Fanuc TP program (LS listing): OP5_LRG_SEQCHNG_AIR_BASE.LS

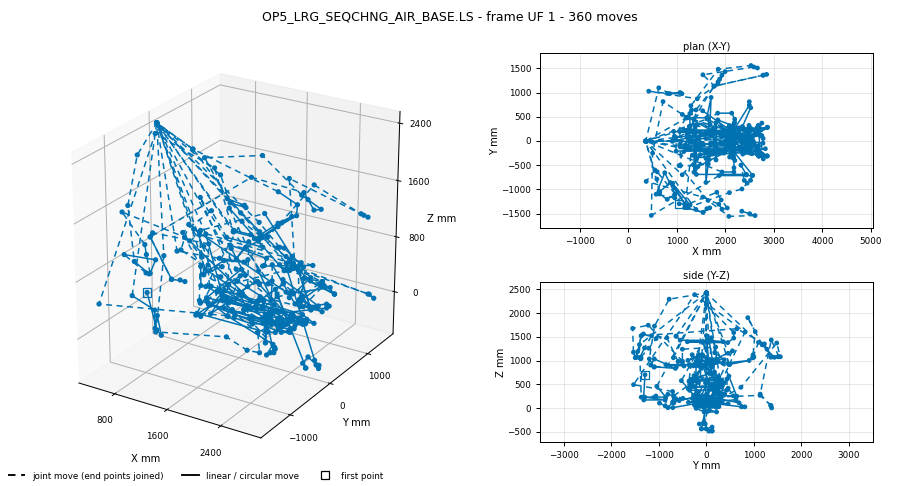
[picture p0: tool path of OP5_LRG_SEQCHNG_AIR_BASE.LS in frame UF 1, 360 of 361 moves have a stored position in this frame; points joined in program order, loops and branches not executed]
/PROG  OP5_LRG_SEQCHNG_AIR_BASE
/ATTR
OWNER		= MNEDITOR;
COMMENT		= "Large Main Air";
PROG_SIZE	= 92875;
CREATE		= DATE 26-02-26  TIME 08:30:24;
MODIFIED	= DATE 26-02-26  TIME 08:30:24;
FILE_NAME	= OP5_LRG_;
VERSION		= 0;
LINE_COUNT	= 2422;
MEMORY_SIZE	= 93511;
PROTECT		= READ_WRITE;
TCD:  STACK_SIZE	= 0,
      TASK_PRIORITY	= 50,
      TIME_SLICE	= 0,
      BUSY_LAMP_OFF	= 0,
      ABORT_REQUEST	= 0,
      PAUSE_REQUEST	= 0;
DEFAULT_GROUP	= 1,1,*,*,*;
CONTROL_CODE	= 00000000 00000000;
/APPL
  ARC Welding Equipment : 1,*,*,*,*;

MPAS ;
MPAS_NUM_PASSES        : 0;
MPAS_LAST_PASS         : 0;
MPAS_CURRENT_PASS      : 0;
MPAS_STATUS_PASS       : 0;
/MN
   1:  !********** WAR HAMMER ********** ;
   2:  !*------- FRAME LARGE ----------* ;
   3:  !*-- WELD SEQUENCE CHANGE 2026--* ;
   4:  !*------- FR500 CELL: A --------* ;
   5:  !******************************** ;
   6:   ;
   7:  CALL HOME    ;
   8:  UFRAME_NUM=1 ;
   9:  DO[17:OFF:WIRE BRAKE]=OFF ;
  10:   ;
  11:  !********POSITIONER MOVE******** ;
  12:J P[1] 85% CNT40    ;
  13:   ;
  14:L P[3] 1000mm/sec CNT40    ;
  15:   ;
  16:  !FR50L1000 ;
  17:  IF R[15]=1002,CALL TECH_HOLD ;
  18:   ;
  19:  !TO SKIP FRONT BUMPER WELDS ;
  20:  CALL ARC_DISABLE_FRONT_BMPR_LRG(0) ;
  21:   ;
  22:   ;
 2:  --eg:PASTE (FR50L1000) ;
  29:   ;
  30:   ;
  31:   ;
  32:L P[8] 800mm/sec CNT30    ;
  33:   ;
  34:L P[9] 1000mm/sec CNT30    ;
  35:   ;
  36:   ;
  37:  !FR50L1001 ;
  38:  IF R[15]=1003,CALL TECH_HOLD ;
  39:   ;
  40:   ;
  41:   ;
 2:  --eg:PASTE (FR50L1001) ;
  48:   ;
  49:   ;
  50:L P[12] 1000mm/sec CNT100    ;
  51:   ;
  52:   ;
  53:  !FR50L1002 ;
  54:  IF R[15]=1004,CALL TECH_HOLD ;
  55:   ;
  56:   ;
  57:L P[13] 1000mm/sec CNT70    ;
  58:   ;
  59:   ;
 2:  --eg:PASTE (FR50L1002) ;
  66:   ;
  67:   ;
  68:  CALL ARC_DISABLE_FRONT_BMPR_LRG(1) ;
  69:   ;
  70:L P[16] 1000mm/sec CNT100    ;
  71:   ;
  72:  !HOME ;
  73:J P[4] 70% CNT30    ;
  74:   ;
  75:  !********POSITIONER MOVE******** ;
  76:J P[17] 85% CNT30    ;
  77:   ;
  78:J P[18] 50% CNT100    ;
  79:   ;
  80:L P[19] 1000mm/sec CNT100    ;
  81:   ;
  82:   ;
  83:  !FR50L1003 ;
  84:  IF R[15]=1005,CALL TECH_HOLD ;
  85:   ;
  86:   ;
  87:L P[20] 1000mm/sec CNT25    ;
  88:   ;
  89:   ;
 2:  --eg:PASTE (FR50L1003) ;
  97:   ;
  98:   ;
  99:L P[24] 1000mm/sec CNT30    ;
 100:   ;
 101:   ;
 102:  !FR50L1010 ;
 103:  IF R[15]=1012,CALL TECH_HOLD ;
 104:   ;
 105:   ;
 106:L P[25] 1000mm/sec CNT30    ;
 107:   ;
 108:   ;
 2:  --eg:PASTE (FR50L1010) ;
 116:   ;
 117:   ;
 118:L P[29] 1000mm/sec CNT25    ;
 119:   ;
 120:   ;
 121:  !FR50L1020 ;
 122:  IF R[15]=1022,CALL TECH_HOLD ;
 123:   ;
 124:   ;
 125:J P[30] 50% CNT25    ;
 126:   ;
 127:   ;
 2:  --eg:PASTE (FR50L1020) ;
 134:   ;
 135:   ;
 136:L P[33] 1000mm/sec CNT30    ;
 137:   ;
 138:L P[34] 1000mm/sec CNT30    ;
 139:   ;
 140:   ;
 141:  !FR50L1030 ;
 142:  IF R[15]=1032,CALL TECH_HOLD ;
 143:   ;
 144:   ;
 145:   ;
 2:  --eg:PASTE (FR50L1030) ;
 152:   ;
 153:   ;
 154:L P[37] 1000mm/sec CNT50    ;
 155:   ;
 156:J P[38] 50% CNT50    ;
 157:   ;
 158:L P[39] 1000mm/sec CNT25    ;
 159:   ;
 160:   ;
 161:  !FR50L1040 ;
 162:  IF R[15]=1042,CALL TECH_HOLD ;
 163:   ;
 164:   ;
 165:   ;
 2:  --eg:PASTE (FR50L1040) ;
 170:   ;
 171:   ;
 172:L P[42] 1000mm/sec CNT30    ;
 173:   ;
 174:L P[43] 1000mm/sec CNT70    ;
 175:   ;
 176:J P[44] 50% CNT50    ;
 177:   ;
 178:L P[45] 1000mm/sec CNT30    ;
 179:   ;
 180:   ;
 181:  !FR50L1050 ;
 182:  IF R[15]=1052,CALL TECH_HOLD ;
 183:   ;
 184:   ;
 185:   ;
 2:  --eg:PASTE (FR50L1050) ;
 190:   ;
 191:   ;
 192:L P[48] 1000mm/sec CNT80    ;
 193:   ;
 194:J P[49] 50% CNT25    ;
 195:   ;
 196:L P[50] 1000mm/sec CNT25    ;
 197:   ;
 198:   ;
 199:  !FR50L1060 ;
 200:  IF R[15]=1062,CALL TECH_HOLD ;
 201:   ;
 202:   ;
 203:   ;
 2:  --eg:PASTE (FR50L1060) ;
 208:   ;
 209:   ;
 210:L P[53] 500mm/sec CNT100    ;
 211:   ;
 212:L P[54] 1500mm/sec CNT35    ;
 213:   ;
 214:J P[55] 50% CNT30    ;
 215:   ;
 216:L P[56] 1000mm/sec CNT30    ;
 217:   ;
 218:   ;
 219:  !FR50L1070 ;
 220:  IF R[15]=1072,CALL TECH_HOLD ;
 221:   ;
 222:   ;
 223:   ;
 2:  --eg:PASTE (FR50L1070) ;
 230:   ;
 231:   ;
 232:L P[59] 1000mm/sec CNT100    ;
 233:   ;
 234:L P[60] 1000mm/sec CNT80    ;
 235:   ;
 236:   ;
 237:  !FR50L1080 ;
 238:  IF R[15]=1082,CALL TECH_HOLD ;
 239:   ;
 240:   ;
 241:   ;
 2:  --eg:PASTE (FR50L1080) ;
 248:   ;
 249:   ;
 250:J P[63] 30% CNT100    ;
 251:   ;
 252:J P[64] 50% CNT100    ;
 253:   ;
 254:L P[65] 1000mm/sec CNT80    ;
 255:   ;
 256:   ;
 257:  !FR50L1090 ;
 258:  IF R[15]=1092,CALL TECH_HOLD ;
 259:  !10MM PASS ;
 260:   ;
 261:   ;
 262:   ;
 2:  --eg:PASTE (FR50L1090) ;
 272:   ;
 273:   ;
 274:J P[72] 16% CNT25    ;
 275:   ;
 276:J P[74] 50% CNT25    ;
 277:   ;
 278:L P[75] 1000mm/sec CNT25    ;
 279:   ;
 280:   ;
 281:  !FR50L1100 ;
 282:  IF R[15]=1102,CALL TECH_HOLD ;
 283:   ;
 284:   ;
 285:   ;
 2:  --eg:PASTE (FR50L1100) ;
 295:   ;
 296:   ;
 297:J P[82] 50% CNT10    ;
 298:   ;
 299:J P[83] 50% CNT80    ;
 300:   ;
 301:L P[84] 1000mm/sec CNT25    ;
 302:   ;
 303:   ;
 304:  !FR50L1110MP1 ;
 305:  IF R[15]=1112,CALL TECH_HOLD ;
 306:   ;
 307:   ;
 308:  MP Offset  PR[3] RPM[1] ;
 309:   ;
 2:  --eg:PASTE (FR50L1110MP1) ;
 317:   ;
 318:  MP Offset End ;
 319:   ;
 320:J P[91] 40% CNT10    ;
 321:   ;
 322:J P[92] 50% CNT30    ;
 323:   ;
 324:L P[93] 1000mm/sec CNT25    ;
 325:   ;
 326:   ;
 327:  !FR50M1110MP2 ;
 328:   ;
 329:   ;
 330:  MP Offset  PR[4] RPM[1] ;
 331:   ;
 2:  --eg:PASTE (FR50M1110MP2) ;
 339:   ;
 340:  MP Offset End ;
 341:   ;
 342:J P[100] 50% CNT25    ;
 343:   ;
 344:J P[102] 50% CNT25    ;
 345:   ;
 346:L P[103] 1000mm/sec CNT25    ;
 347:   ;
 348:   ;
 349:  !FR50L1120MP3 ;
 350:  IF R[15]=1122,CALL TECH_HOLD ;
 351:   ;
 352:   ;
 353:  MP Offset  PR[1] RPM[2] ;
 354:   ;
 2:  --eg:PASTE (FR50L1120MP3) ;
 362:   ;
 363:  MP Offset End ;
 364:   ;
 365:J P[110] 50% CNT25    ;
 366:   ;
 367:J P[111] 50% CNT25    ;
 368:   ;
 369:L P[112] 1000mm/sec CNT25    ;
 370:   ;
 371:   ;
 372:  !FR501130MP4 ;
 373:   ;
 374:   ;
 375:  MP Offset  PR[2] RPM[2] ;
 376:   ;
 2:  --eg:PASTE (FR501130MP4) ;
 384:   ;
 385:  MP Offset End ;
 386:   ;
 387:J P[119] 50% CNT25    ;
 388:   ;
 389:J P[121] 50% CNT25    ;
 390:   ;
 391:L P[122] 1000mm/sec CNT25    ;
 392:   ;
 393:   ;
 394:  !FR50L1140 ;
 395:  IF R[15]=1142,CALL TECH_HOLD ;
 396:   ;
 397:   ;
 398:   ;
 2:  --eg:PASTE (FR50L1140) ;
 404:   ;
 405:   ;
 406:L P[127] 1000mm/sec CNT25    ;
 407:   ;
 408:J P[128] 50% CNT25    ;
 409:   ;
 410:   ;
 411:  !FR50L1141 ;
 412:  IF R[15]=1143,CALL TECH_HOLD ;
 413:   ;
 414:   ;
 415:   ;
 2:  --eg:PASTE (FR50L1141) ;
 421:   ;
 422:   ;
 423:L P[133] 1000mm/sec CNT25    ;
 424:   ;
 425:L P[134] 1000mm/sec CNT25    ;
 426:   ;
 427:J P[135] 50% CNT25    ;
 428:   ;
 429:L P[136] 1000mm/sec CNT50    ;
 430:   ;
 431:   ;
 432:  !FR50L1150 ;
 433:  IF R[15]=1152,CALL TECH_HOLD ;
 434:   ;
 435:   ;
 436:   ;
 2:  --eg:PASTE (FR50L1150) ;
 443:   ;
 444:   ;
 445:L P[139] 1000mm/sec CNT100    ;
 446:   ;
 447:L P[140] 1000mm/sec CNT50    ;
 448:   ;
 449:   ;
 450:  !FR50L1160 ;
 451:  IF R[15]=1162,CALL TECH_HOLD ;
 452:   ;
 453:   ;
 2:  --eg:PASTE (FR50L1160) ;
 460:   ;
 461:   ;
 462:L P[143] 1000mm/sec CNT30    ;
 463:   ;
 464:  !********POSITIONER MOVE******** ;
 465:J P[144] 85% CNT30    ;
 466:   ;
 467:L P[145] 1000mm/sec CNT100    ;
 468:   ;
 469:   ;
 470:  !FR50L1170 ;
 471:  IF R[15]=1172,CALL TECH_HOLD ;
 472:   ;
 473:   ;
 474:   ;
 2:  --eg:PASTE (FR50L1170) ;
 481:   ;
 482:   ;
 483:L P[148] 1000mm/sec CNT100    ;
 484:   ;
 485:L P[149] 1500mm/sec CNT100    ;
 486:   ;
 487:   ;
 488:  !FR50L1180 ;
 489:  IF R[15]=1182,CALL TECH_HOLD ;
 490:   ;
 491:   ;
 492:   ;
 2:  --eg:PASTE (FR50L1180) ;
 499:   ;
 500:   ;
 501:L P[152] 1000mm/sec CNT100    ;
 502:   ;
 503:  !HOME ;
 504:J P[7] 100% CNT30    ;
 505:   ;
 506:  !********POSITIONER MOVE******** ;
 507:J P[153] 80% CNT30    ;
 508:   ;
 509:J P[154] 50% CNT100    ;
 510:   ;
 511:L P[155] 1000mm/sec CNT25    ;
 512:   ;
 513:   ;
 514:  !FR50L1210 ;
 515:  IF R[15]=1212,CALL TECH_HOLD ;
 516:   ;
 517:   ;
 518:   ;
 2:  --eg:PASTE (FR50L1210) ;
 526:   ;
 527:   ;
 528:L P[159] 1000mm/sec CNT25    ;
 529:   ;
 530:L P[160] 1000mm/sec CNT25    ;
 531:   ;
 532:   ;
 533:  !FR50L1220 ;
 534:  IF R[15]=1222,CALL TECH_HOLD ;
 535:   ;
 536:   ;
 537:   ;
 2:  --eg:PASTE (FR50L1220) ;
 544:   ;
 545:   ;
 546:L P[163] 1000mm/sec CNT80    ;
 547:   ;
 548:L P[164] 1200mm/sec CNT25    ;
 549:   ;
 550:   ;
 551:  !FR50L1230 ;
 552:  IF R[15]=1232,CALL TECH_HOLD ;
 553:   ;
 554:   ;
 555:   ;
 2:  --eg:PASTE (FR50L1230) ;
 562:   ;
 563:   ;
 564:L P[167] 1000mm/sec CNT25    ;
 565:   ;
 566:L P[168] 1000mm/sec CNT25    ;
 567:   ;
 568:   ;
 569:  !FR50L1240 ;
 570:  IF R[15]=1242,CALL TECH_HOLD ;
 571:   ;
 572:   ;
 573:   ;
 2:  --eg:PASTE (FR50L1240) ;
 581:   ;
 582:   ;
 583:L P[172] 1000mm/sec CNT25    ;
 584:   ;
 585:L P[173] 1000mm/sec CNT100    ;
 586:   ;
 587:  !HOME ;
 588:J P[116] 100% CNT100    ;
 589:   ;
 590:   ;
 591:  !********POSITIONER MOVE******** ;
 592:J P[174] 85% FINE    ;
 593:   ;
 594:  CALL T_CLEAN    ;
 595:   ;
 596:J P[175] 50% CNT35    ;
 597:   ;
 598:L P[176] 1000mm/sec CNT25    ;
 599:   ;
 600:   ;
 601:  !FR50L1250 ;
 602:  IF R[15]=1252,CALL TECH_HOLD ;
 603:   ;
 604:   ;
 605:   ;
 2:  --eg:PASTE (FR50L1250) ;
 614:   ;
 615:   ;
 616:L P[181] 1000mm/sec CNT100    ;
 617:   ;
 618:J P[182] 50% CNT100    ;
 619:   ;
 620:L P[184] 500mm/sec CNT100    ;
 621:   ;
 622:   ;
 623:  !FR50L1260 ;
 624:  IF R[15]=1262,CALL TECH_HOLD ;
 625:   ;
 626:   ;
 627:   ;
 2:  --eg:PASTE (FR50L1260) ;
 636:   ;
 637:   ;
 638:L P[189] 1000mm/sec CNT25    ;
 639:   ;
 640:J P[190] 50% CNT25    ;
 641:   ;
 642:L P[191] 1000mm/sec CNT25    ;
 643:   ;
 644:   ;
 645:  !FR50L1270 ;
 646:  IF R[15]=1272,CALL TECH_HOLD ;
 647:   ;
 648:   ;
 649:   ;
 2:  --eg:PASTE (FR50L1270) ;
 657:   ;
 658:   ;
 659:L P[195] 1000mm/sec CNT80    ;
 660:   ;
 661:L P[196] 1000mm/sec CNT100    ;
 662:   ;
 663:   ;
 664:  !FR50L1280 ;
 665:  IF R[15]=1282,CALL TECH_HOLD ;
 666:   ;
 667:   ;
 668:   ;
 2:  --eg:PASTE (FR50L1280) ;
 676:   ;
 677:   ;
 678:L P[200] 1000mm/sec CNT25    ;
 679:   ;
 680:J P[201] 50% CNT25    ;
 681:   ;
 682:L P[202] 1000mm/sec CNT25    ;
 683:   ;
 684:   ;
 685:  !FR50L1290 ;
 686:  IF R[15]=1292,CALL TECH_HOLD ;
 687:   ;
 688:   ;
 689:   ;
 2:  --eg:PASTE (FR50L1290) ;
 697:   ;
 698:   ;
 699:L P[206] 1000mm/sec CNT100    ;
 700:   ;
 701:L P[207] 1000mm/sec CNT100    ;
 702:   ;
 703:   ;
 704:  !FR50L1300 ;
 705:  IF R[15]=1302,CALL TECH_HOLD ;
 706:   ;
 707:   ;
 708:   ;
 2:  --eg:PASTE (FR50L1300) ;
 715:   ;
 716:   ;
 717:L P[210] 1000mm/sec CNT100    ;
 718:   ;
 719:L P[211] 1000mm/sec CNT100    ;
 720:   ;
 721:   ;
 722:  !FR50L1310 ;
 723:  IF R[15]=1312,CALL TECH_HOLD ;
 724:   ;
 725:   ;
 726:   ;
 2:  --eg:PASTE (FR50L1310) ;
 733:   ;
 734:   ;
 735:L P[214] 1000mm/sec CNT100    ;
 736:   ;
 737:L P[215] 1000mm/sec CNT100    ;
 738:   ;
 739:   ;
 740:  !FR50L1320 ;
 741:  IF R[15]=1322,CALL TECH_HOLD ;
 742:   ;
 743:   ;
 744:   ;
 2:  --eg:PASTE (FR50L1320) ;
 752:   ;
 753:   ;
 754:L P[219] 1000mm/sec CNT100    ;
 755:   ;
 756:L P[220] 1000mm/sec CNT100    ;
 757:   ;
 758:J P[73] 50% CNT30    ;
 759:   ;
 760:  !********POSITIONER MOVE******** ;
 761:J P[86] 100% CNT30    ;
 762:   ;
 763:  !FR50L1330 ;
 764:  IF R[15]=1332,CALL TECH_HOLD ;
 765:   ;
 766:   ;
 767:J P[327] 40% CNT10    ;
 768:   ;
 769:   ;
 2:  --eg:PASTE (FR50L1330) ;
 774:   ;
 775:   ;
 776:J P[85] 50% CNT30    ;
 777:   ;
 778:L P[233] 1000mm/sec CNT25    ;
 779:   ;
 780:  !********POSITIONER MOVE******** ;
 781:J P[225] 80% CNT20    ;
 782:   ;
 783:   ;
 784:   ;
 785:  !FR50L1340 ;
 786:  IF R[15]=1342,CALL TECH_HOLD ;
 787:   ;
 788:   ;
 789:   ;
 2:  --eg:PASTE (FR50L1340) ;
 794:   ;
 795:   ;
 796:   ;
 797:  !FR50L1350 ;
 798:  IF R[15]=1352,CALL TECH_HOLD ;
 799:   ;
 800:   ;
 801:   ;
 2:  --eg:PASTE (FR50L1350) ;
 806:   ;
 807:   ;
 808:L P[230] 1000mm/sec CNT25    ;
 809:   ;
 810:  !HOME ;
 811:J P[117] 100% CNT50    ;
 812:   ;
 813:  !********POSITIONER MOVE******** ;
 814:J P[768] 85% CNT25    ;
 815:   ;
 816:L P[234] 1000mm/sec CNT25    ;
 817:   ;
 818:J P[235] 50% CNT25    ;
 819:   ;
 820:   ;
 821:  !FR50L1380 ;
 822:  IF R[15]=1382,CALL TECH_HOLD ;
 823:   ;
 824:   ;
 825:   ;
 2:  --eg:PASTE (FR50L1380) ;
 834:   ;
 835:   ;
 836:L P[240] 800mm/sec CNT2    ;
 837:   ;
 838:L P[241] 800mm/sec CNT25    ;
 839:   ;
 840:  !********POSITIONER MOVE******** ;
 841:J P[242] 75% CNT5    ;
 842:   ;
 843:L P[243] 1000mm/sec CNT25    ;
 844:   ;
 845:   ;
 846:  !FR50L1390 ;
 847:  IF R[15]=1392,CALL TECH_HOLD ;
 848:   ;
 849:   ;
 2:  --eg:PASTE (FR50L1390) ;
 856:   ;
 857:   ;
 858:L P[248] 1000mm/sec CNT25    ;
 859:   ;
 860:L P[249] 1000mm/sec CNT25    ;
 861:   ;
 862:   ;
 863:  !FR50L1400 ;
 864:  IF R[15]=1402,CALL TECH_HOLD ;
 865:   ;
 866:   ;
 867:   ;
 2:  --eg:PASTE (FR50L1400) ;
 874:   ;
 875:   ;
 876:L P[252] 1000mm/sec CNT25    ;
 877:   ;
 878:   ;
 879:  !FR50L1410 ;
 880:  IF R[15]=1412,CALL TECH_HOLD ;
 881:   ;
 882:   ;
 883:   ;
 2:  --eg:PASTE (FR50L1410) ;
 891:   ;
 892:   ;
 893:L P[256] 1000mm/sec CNT25    ;
 894:   ;
 895:   ;
 896:  !FR50L1420 ;
 897:  IF R[15]=1422,CALL TECH_HOLD ;
 898:   ;
 899:   ;
 900:   ;
 2:  --eg:PASTE (FR50L1420) ;
 908:   ;
 909:   ;
 910:L P[260] 1000mm/sec CNT25    ;
 911:   ;
 912:L P[261] 1000mm/sec CNT25    ;
 913:   ;
 914:   ;
 915:  !FR50L1430 ;
 916:  IF R[15]=1432,CALL TECH_HOLD ;
 917:   ;
 918:   ;
 919:   ;
 2:  --eg:PASTE (FR50L1430) ;
 925:   ;
 926:   ;
 927:L P[265] 1000mm/sec CNT25    ;
 928:   ;
 929:   ;
 930:  !FR50L1431 ;
 931:  IF R[15]=1433,CALL TECH_HOLD ;
 932:   ;
 933:   ;
 934:   ;
 2:  --eg:PASTE (FR50L1431) ;
 940:   ;
 941:   ;
 942:L P[269] 1000mm/sec CNT25    ;
 943:   ;
 944:L P[270] 1000mm/sec CNT25    ;
 945:   ;
 946:L P[271] 1000mm/sec CNT50 Wjnt    ;
 947:   ;
 948:J P[272] 50% CNT25    ;
 949:   ;
 950:L P[273] 1000mm/sec CNT25    ;
 951:   ;
 952:   ;
 953:  !FR50L1440 ;
 954:  IF R[15]=1442,CALL TECH_HOLD ;
 955:   ;
 956:   ;
 957:   ;
 2:  --eg:PASTE (FR50L1440) ;
 964:   ;
 965:   ;
 966:L P[276] 1000mm/sec CNT25    ;
 967:   ;
 968:   ;
 969:  !FR50L1450 ;
 970:  IF R[15]=1452,CALL TECH_HOLD ;
 971:   ;
 972:   ;
 973:   ;
 2:  --eg:PASTE (FR50L1450) ;
 981:   ;
 982:   ;
 983:L P[280] 1000mm/sec CNT25    ;
 984:   ;
 985:L P[281] 1000mm/sec CNT25    ;
 986:   ;
 987:   ;
 988:  !FR50L1460 ;
 989:  IF R[15]=1462,CALL TECH_HOLD ;
 990:   ;
 991:   ;
 992:   ;
 2:  --eg:PASTE (FR50L1460) ;
1000:   ;
1001:   ;
1002:L P[285] 1000mm/sec CNT25    ;
1003:   ;
1004:  !********POSITIONER MOVE******** ;
1005:J P[286] 75% CNT15    ;
1006:   ;
1007:L P[287] 1000mm/sec CNT25    ;
1008:   ;
1009:   ;
1010:  !FR50L1470 ;
1011:  IF R[15]=1472,CALL TECH_HOLD ;
1012:   ;
1013:   ;
1014:   ;
 2:  --eg:PASTE (FR50L1470) ;
1021:   ;
1022:   ;
1023:L P[290] 1000mm/sec CNT25    ;
1024:   ;
1025:  !********POSITIONER MOVE******** ;
1026:J P[291] 85% CNT2    ;
1027:   ;
1028:L P[292] 1000mm/sec CNT25    ;
1029:   ;
1030:   ;
1031:  !FR50L1480 ;
1032:  IF R[15]=1482,CALL TECH_HOLD ;
1033:   ;
1034:   ;
1035:   ;
 2:  --eg:PASTE (FR50L1480) ;
1040:   ;
1041:   ;
1042:L P[295] 1000mm/sec CNT25    ;
1043:   ;
1044:L P[296] 1000mm/sec CNT25    ;
1045:   ;
1046:   ;
1047:  !FR50L1490 ;
1048:  IF R[15]=1492,CALL TECH_HOLD ;
1049:   ;
1050:   ;
1051:   ;
 2:  --eg:PASTE (FR50L1490) ;
1058:   ;
1059:   ;
1060:L P[299] 1000mm/sec CNT25    ;
1061:   ;
1062:L P[300] 1000mm/sec CNT25    ;
1063:   ;
1064:L P[301] 1000mm/sec CNT25    ;
1065:   ;
1066:  !********POSITIONER MOVE******** ;
1067:J P[302] 85% FINE    ;
1068:   ;
1069:L P[303] 1000mm/sec CNT25    ;
1070:   ;
1071:   ;
1072:  !FR50L1500 ;
1073:  IF R[15]=1502,CALL TECH_HOLD ;
1074:   ;
1075:   ;
1076:   ;
 2:  --eg:PASTE (FR50L1500) ;
1082:   ;
1083:   ;
1084:L P[307] 1000mm/sec CNT25    ;
1085:   ;
1086:J P[308] 50% CNT25    ;
1087:   ;
1088:L P[309] 1000mm/sec CNT25    ;
1089:   ;
1090:   ;
1091:  !FR50L1510 ;
1092:  IF R[15]=1512,CALL TECH_HOLD ;
1093:   ;
1094:   ;
1095:   ;
 2:  --eg:PASTE (FR50L1510) ;
1108:   ;
1109:L P[321] 1000mm/sec CNT80    ;
1110:   ;
1111:J P[322] 40% CNT80    ;
1112:   ;
1113:  --eg:Insert g2j2 @90 Loadstop!!! ;
1116:   ;
1117:  !********POSITIONER MOVE******** ;
1118:J P[114] 85% CNT40    ;
1119:   ;
1120:J P[115] 50% CNT25    ;
1121:   ;
1122:  CALL ARC_DISABLE_RH_LS(0) ;
1123:   ;
1124:   ;
1125:  !FR50L2040 ;
1126:  IF R[15]=2042,CALL TECH_HOLD ;
1127:   ;
1128:   ;
1129:L P[473] 1000mm/sec CNT25    ;
1130:   ;
1131:   ;
 2:  --eg:PASTE (FR50L2040) ;
1141:   ;
1142:  CALL ARC_DISABLE_RH_LS(1) ;
1143:   ;
1144:L P[494] 1000mm/sec CNT25    ;
1145:   ;
1146:J P[497] 50% CNT75    ;
1147:   ;
1148:  --eg:Insert g2j2 @90 Loadstop!!! ;
1151:   ;
1152:   ;
1153:   ;
1154:  !********POSITIONER MOVE******** ;
1155:J P[502] 40% CNT40    ;
1156:   ;
1157:J P[323] 40% CNT25    ;
1158:   ;
1159:  !CELL ID: A . ;
1160:   ;
 2:  --eg:PASTE (FRID) ;
1163:   ;
1164:J P[324] 50% CNT30    ;
1165:   ;
1166:L P[328] 800mm/sec CNT60    ;
1167:   ;
1168:J P[224] 40% CNT100    ;
1169:   ;
1170:J P[329] 40% CNT90    ;
1171:   ;
1172:J P[331] 50% CNT50    ;
1173:   ;
1174:L P[332] 1000mm/sec CNT25    ;
1175:   ;
1176:   ;
1177:  !FR50L1520 ;
1178:  IF R[15]=1522,CALL TECH_HOLD ;
1179:   ;
1180:   ;
1181:   ;
 2:  --eg:PASTE (FR50L1520) ;
1188:   ;
1189:   ;
1190:L P[335] 1000mm/sec CNT25    ;
1191:   ;
1192:J P[336] 50% CNT25    ;
1193:   ;
1194:L P[337] 1000mm/sec CNT25    ;
1195:   ;
1196:   ;
1197:  !FR50L1530 ;
1198:  IF R[15]=1532,CALL TECH_HOLD ;
1199:   ;
1200:   ;
1201:   ;
 2:  --eg:PASTE (FR50L1530) ;
1208:   ;
1209:   ;
1210:L P[340] 1000mm/sec CNT25    ;
1211:   ;
1212:L P[341] 1000mm/sec CNT25    ;
1213:   ;
1214:L P[342] 1000mm/sec CNT25    ;
1215:   ;
1216:  !FR50L1540 ;
1217:  IF R[15]=1542,CALL TECH_HOLD ;
1218:   ;
1219:   ;
 2:  --eg:PASTE (FR50L1540) ;
1227:   ;
1228:L P[346] 1000mm/sec CNT40    ;
1229:   ;
1230:L P[347] 1100mm/sec CNT50 Wjnt    ;
1231:   ;
1232:J P[348] 50% CNT35    ;
1233:   ;
1234:  --eg:Insert g2j2 @90 content ;
1236:   ;
1237:J P[88] 50% CNT90    ;
1238:   ;
1239:L P[96] 1000mm/sec CNT25    ;
1240:   ;
1241:   ;
1242:  !FR50L1590 ;
1243:  IF R[15]=1592,CALL TECH_HOLD ;
1244:   ;
1245:   ;
1246:   ;
 2:  --eg:PASTE (FR50L1590) ;
1253:   ;
1254:   ;
1255:L P[120] 1000mm/sec CNT25    ;
1256:   ;
1257:J P[123] 50% CNT25    ;
1258:   ;
1259:   ;
1260:  !FR50L1600 ;
1261:  IF R[15]=1602,CALL TECH_HOLD ;
1262:   ;
1263:   ;
1264:   ;
 2:  --eg:PASTE (FR50L1600) ;
1271:   ;
1272:   ;
1273:L P[126] 1000mm/sec CNT25    ;
1274:   ;
1275:J P[129] 50% CNT25    ;
1276:   ;
1277:   ;
1278:  !FR50L1601 ;
1279:  IF R[15]=1603,CALL TECH_HOLD ;
1280:   ;
1281:   ;
1282:   ;
 2:  --eg:PASTE (FR50L1601) ;
1289:   ;
1290:   ;
1291:L P[132] 1000mm/sec CNT25    ;
1292:   ;
1293:L P[137] 1200mm/sec CNT40 Wjnt    ;
1294:   ;
1295:  !********POSITIONER MOVE******** ;
1296:J P[138] 90% CNT30    ;
1297:   ;
1298:L P[141] 1000mm/sec CNT25    ;
1299:   ;
1300:L P[142] 1000mm/sec CNT25    ;
1301:   ;
1302:   ;
1303:  !FR50L1610 ;
1304:  IF R[15]=1612,CALL TECH_HOLD ;
1305:   ;
1306:   ;
1307:   ;
 2:  --eg:PASTE (FR50L1610) ;
1315:   ;
1316:   ;
1317:L P[151] 1000mm/sec CNT25    ;
1318:   ;
1319:L P[156] 1000mm/sec CNT25    ;
1320:   ;
1321:   ;
1322:   ;
1323:  !FR50L1620 ;
1324:  IF R[15]=1622,CALL TECH_HOLD ;
1325:   ;
1326:   ;
1327:   ;
 2:  --eg:PASTE (FR50L1620) ;
1335:   ;
1336:   ;
1337:L P[365] 1000mm/sec CNT75    ;
1338:   ;
1339:L P[376] 1000mm/sec CNT25    ;
1340:   ;
1341:J P[380] 50% CNT40    ;
1342:   ;
1343:  !********POSITIONER MOVE******** ;
1344:J P[504] 85% CNT30    ;
1345:   ;
1346:  CALL HOME    ;
1347:  CALL T_CLEAN    ;
1348:   ;
1349:J P[381] 90% CNT30    ;
1350:   ;
1351:J P[397] 50% CNT25    ;
1352:   ;
1353:   ;
1354:  !FR50L1630 ;
1355:  IF R[15]=1632,CALL TECH_HOLD ;
1356:   ;
1357:   ;
1358:   ;
 2:  --eg:PASTE (FR50L1630) ;
1369:   ;
1370:   ;
1371:L P[412] 1000mm/sec CNT40    ;
1372:   ;
1373:J P[413] 50% CNT35    ;
1374:   ;
1375:   ;
1376:  !FR50L1640 ;
1377:  IF R[15]=1642,CALL TECH_HOLD ;
1378:   ;
1379:   ;
1380:   ;
 2:  --eg:PASTE (FR50L1640) ;
1393:   ;
1394:   ;
1395:L P[432] 1000mm/sec CNT100    ;
1396:   ;
1397:J P[433] 50% CNT35    ;
1398:   ;
1399:  !********POSITIONER MOVE******** ;
1400:J P[434] 85% CNT30    ;
1401:   ;
1402:L P[435] 1000mm/sec CNT25    ;
1403:   ;
1404:J P[436] 50% CNT25    ;
1405:   ;
1406:   ;
1407:  !FR50L1650 ;
1408:  IF R[15]=1652,CALL TECH_HOLD ;
1409:   ;
1410:   ;
1411:   ;
 2:  --eg:PASTE (FR50L1650) ;
1428:   ;
1429:   ;
1430:L P[451] 1000mm/sec CNT100    ;
1431:   ;
1432:L P[452] 1000mm/sec CNT80    ;
1433:   ;
1434:   ;
1435:  !FR50L1651 ;
1436:  IF R[15]=1653,CALL TECH_HOLD ;
1437:   ;
1438:   ;
1439:   ;
 2:  --eg:PASTE (FR50L1651) ;
1448:   ;
1449:   ;
1450:L P[459] 1000mm/sec CNT60    ;
1451:   ;
1452:L P[460] 1000mm/sec CNT100    ;
1453:   ;
1454:J P[461] 50% CNT40    ;
1455:   ;
1456:J P[498] 50% CNT40    ;
1457:  --eg:Insert g2j2 @90 content ;
1458:   ;
1459:  !********POSITIONER MOVE******** ;
1460:J P[350] 90% CNT40    ;
1461:   ;
1462:J P[349] 50% CNT25    ;
1463:   ;
1464:L P[351] 1000mm/sec CNT25    ;
1465:   ;
1466:   ;
1467:  !FR50L1540 ;
1468:  IF R[15]=1542,CALL TECH_HOLD ;
1469:   ;
1470:   ;
1471:   ;
 2:  --eg:PASTE (FR50L1540) ;
1484:   ;
1485:   ;
1486:L P[360] 1000mm/sec CNT60    ;
1487:   ;
1488:L P[361] 1000mm/sec CNT25    ;
1489:   ;
1490:   ;
1491:  !FR50L1550 ;
1492:  IF R[15]=1552,CALL TECH_HOLD ;
1493:   ;
1494:   ;
1495:   ;
 2:  --eg:PASTE (FR50L1550) ;
1505:   ;
1506:   ;
1507:L P[367] 1000mm/sec CNT25    ;
1508:   ;
1509:L P[368] 1000mm/sec CNT40    ;
1510:   ;
1511:J P[183] 50% CNT40    ;
1512:   ;
1513:  !********POSITIONER MOVE******** ;
1514:J P[377] 90% CNT30    ;
1515:   ;
1516:J P[378] 50% CNT40    ;
1517:   ;
1518:J P[379] 50% CNT40    ;
1519:   ;
1520:   ;
1521:  !FR50L1570 ;
1522:  IF R[15]=1572,CALL TECH_HOLD ;
1523:   ;
1524:   ;
1525:   ;
 2:  --eg:PASTE (FR50L1570) ;
1538:   ;
1539:   ;
1540:L P[388] 1000mm/sec CNT100    ;
1541:   ;
1542:L P[389] 1000mm/sec CNT25    ;
1543:   ;
1544:   ;
1545:  !FR50L1580 ;
1546:  IF R[15]=1582,CALL TECH_HOLD ;
1547:   ;
1548:   ;
1549:   ;
 2:  --eg:PASTE (FR50L1580) ;
1559:   ;
1560:   ;
1561:L P[395] 600mm/sec CNT25    ;
1562:   ;
1563:L P[396] 1000mm/sec CNT100    ;
1564:   ;
1565:J P[326] 60% CNT25    ;
1566:   ;
1567:J P[325] 70% CNT30    ;
1568:   ;
1569:  !********POSITIONER MOVE******** ;
1570:J P[503] 90% CNT30    ;
1571:   ;
1572:J P[477] 50% CNT40    ;
1573:   ;
1574:J P[478] 50% CNT80    ;
1575:   ;
1576:J P[479] 50% CNT60    ;
1577:   ;
1578:J P[480] 50% CNT30    ;
1579:   ;
1580:   ;
1581:  !FR50L1660 ;
1582:  IF R[15]=1662,CALL TECH_HOLD ;
1583:   ;
1584:   ;
1585:   ;
 2:  --eg:PASTE (FR50L1660) ;
1592:   ;
1593:   ;
1594:J P[483] 20% CNT100    ;
1595:   ;
1596:J P[484] 60% CNT25    ;
1597:   ;
1598:L P[485] 600mm/sec CNT25    ;
1599:   ;
1600:   ;
1601:  !FR50L1661 ;
1602:  IF R[15]=1663,CALL TECH_HOLD ;
1603:   ;
1604:   ;
1605:   ;
 2:  --eg:PASTE (FR50L1661) ;
1612:   ;
1613:   ;
1614:L P[488] 500mm/sec CNT25    ;
1615:   ;
1616:L P[489] 500mm/sec CNT35    ;
1617:   ;
1618:L P[490] 1000mm/sec CNT25    ;
1619:   ;
1620:  !********POSITIONER MOVE******** ;
1621:J P[491] 90% CNT25    ;
1622:   ;
1623:L P[492] 1000mm/sec CNT25    ;
1624:   ;
1625:   ;
1626:  !FR50L1670 ;
1627:  IF R[15]=1672,CALL TECH_HOLD ;
1628:   ;
1629:   ;
1630:   ;
 2:  --eg:PASTE (FR50L1670) ;
1635:   ;
1636:   ;
1637:L P[495] 800mm/sec CNT25    ;
1638:   ;
1639:L P[496] 1000mm/sec CNT25    ;
1640:   ;
1641:   ;
1642:  !FR50L1680 ;
1643:  IF R[15]=1682,CALL TECH_HOLD ;
1644:   ;
1645:   ;
1646:   ;
 2:  --eg:PASTE (FR50L1680) ;
1653:   ;
1654:   ;
1655:L P[499] 1000mm/sec CNT25    ;
1656:   ;
1657:  !********POSITIONER MOVE******** ;
1658:J P[500] 75% CNT20    ;
1659:   ;
1660:L P[501] 1000mm/sec CNT25    ;
1661:   ;
1662:   ;
1663:  !FR50L1690 ;
1664:  IF R[15]=1692,CALL TECH_HOLD ;
1665:   ;
1666:   ;
1667:   ;
 2:  --eg:PASTE (FR50L1690) ;
1675:   ;
1676:   ;
1677:L P[505] 300mm/sec CNT40    ;
1678:   ;
1679:L P[506] 1000mm/sec CNT40    ;
1680:   ;
1681:L P[507] 1000mm/sec CNT40    ;
1682:   ;
1683:   ;
1684:  !FR50L1700 ;
1685:  IF R[15]=1702,CALL TECH_HOLD ;
1686:   ;
1687:   ;
1688:   ;
 2:  --eg:PASTE (FR50L1700) ;
1701:   ;
1702:   ;
1703:L P[519] 1000mm/sec CNT100    ;
1704:   ;
1705:L P[520] 1000mm/sec CNT40    ;
1706:   ;
1707:L P[521] 500mm/sec CNT30    ;
1708:   ;
1709:   ;
1710:  !FR50L1710 ;
1711:  IF R[15]=1712,CALL TECH_HOLD ;
1712:   ;
1713:   ;
1714:   ;
 2:  --eg:PASTE (FR50L1710) ;
1722:   ;
1723:   ;
1724:L P[525] 500mm/sec CNT25    ;
1725:   ;
1726:L P[526] 800mm/sec CNT50 Wjnt    ;
1727:   ;
1728:L P[527] 1400mm/sec CNT100 Wjnt    ;
1729:   ;
1730:J P[528] 50% CNT100    ;
1731:   ;
1732:L P[529] 1000mm/sec CNT25    ;
1733:   ;
1734:   ;
1735:  !FR50L1720 ;
1736:  IF R[15]=1722,CALL TECH_HOLD ;
1737:   ;
1738:   ;
1739:   ;
 2:  --eg:PASTE (FR50L1720) ;
1746:   ;
1747:   ;
1748:J P[534] 50% CNT10    ;
1749:   ;
1750:  !********POSITIONER MOVE******** ;
1751:J P[535] 40% CNT10    ;
1752:   ;
1753:J P[536] 20% CNT5    ;
1754:   ;
1755:L P[537] 1000mm/sec CNT25    ;
1756:   ;
1757:   ;
1758:  !FR50L1730 ;
1759:  IF R[15]=1732,CALL TECH_HOLD ;
1760:   ;
1761:   ;
1762:   ;
 2:  --eg:PASTE (FR50L1730) ;
1771:   ;
1772:   ;
1773:L P[542] 1000mm/sec CNT25    ;
1774:   ;
1775:J P[543] 50% CNT10    ;
1776:   ;
1777:  !********POSITIONER MOVE******** ;
1778:J P[544] 80% CNT10    ;
1779:   ;
1780:   ;
1781:  !FR50L1740 ;
1782:  IF R[15]=1742,CALL TECH_HOLD ;
1783:   ;
1784:   ;
1785:   ;
 2:  --eg:PASTE (FR50L1740) ;
1792:   ;
1793:   ;
1794:L P[547] 1000mm/sec CNT25    ;
1795:   ;
1796:L P[548] 1000mm/sec CNT25    ;
1797:   ;
1798:L P[549] 1000mm/sec CNT25    ;
1799:   ;
1800:   ;
1801:  !FR50L1750 ;
1802:  IF R[15]=1752,CALL TECH_HOLD ;
1803:   ;
1804:   ;
1805:   ;
 2:  --eg:PASTE (FR50L1750) ;
1813:   ;
1814:   ;
1815:L P[553] 1000mm/sec CNT25    ;
1816:   ;
1817:L P[554] 1000mm/sec CNT100    ;
1818:   ;
1819:L P[555] 1000mm/sec CNT100    ;
1820:   ;
1821:J P[508] 50% CNT40    ;
1822:   ;
1823:  CALL HOME    ;
1824:  CALL T_CLEAN    ;
1825:   ;
1826:J P[556] 50% CNT30    ;
1827:   ;
1828:   ;
1829:  !FR50L1770 ;
1830:  IF R[15]=1772,CALL TECH_HOLD ;
1831:   ;
1832:   ;
1833:   ;
 2:  --eg:PASTE (FR50L1770) ;
1840:   ;
1841:   ;
1842:L P[559] 1000mm/sec CNT100    ;
1843:   ;
1844:J P[560] 50% CNT25    ;
1845:   ;
 2:  --eg:PASTE (FR50L1771) ;
1850:L P[563] 1200mm/sec CNT100    ;
1851:   ;
1852:L P[89] 800mm/sec CNT100    ;
1853:   ;
1854:L P[565] 1000mm/sec CNT20    ;
1855:   ;
 2:  --eg:PASTE (FR50L1772) ;
1860:   ;
1861:L P[568] 1000mm/sec CNT25    ;
1862:   ;
1863:J P[569] 50% CNT40    ;
1864:   ;
1865:  !********POSITIONER MOVE******** ;
1866:J P[371] 90% CNT40    ;
1867:   ;
1868:L P[572] 1000mm/sec CNT25    ;
1869:   ;
1870:L P[573] 1000mm/sec CNT25    ;
1871:   ;
1872:   ;
1873:  !FR50L1780 ;
1874:  IF R[15]=1782,CALL TECH_HOLD ;
1875:   ;
1876:   ;
1877:   ;
 2:  --eg:PASTE (FR50L1780) ;
1884:   ;
1885:   ;
1886:L P[576] 500mm/sec CNT25    ;
1887:   ;
1888:L P[577] 1000mm/sec CNT25    ;
1889:   ;
1890:  !********POSITIONER MOVE******** ;
1891:J P[578] 90% CNT25    ;
1892:   ;
1893:   ;
1894:  !FR50L1790 ;
1895:  IF R[15]=1792,CALL TECH_HOLD ;
1896:   ;
1897:   ;
1898:   ;
 2:  --eg:PASTE (FR50L1790) ;
1905:   ;
1906:   ;
1907:L P[581] 1000mm/sec CNT100    ;
1908:   ;
1909:   ;
1910:  !FR50L1800 ;
1911:  IF R[15]=1802,CALL TECH_HOLD ;
1912:   ;
1913:   ;
1914:   ;
 2:  --eg:PASTE (FR50L1800) ;
1922:   ;
1923:   ;
1924:L P[585] 1000mm/sec CNT40    ;
1925:   ;
1926:   ;
1927:  !FR50L1810 ;
1928:  IF R[15]=1812,CALL TECH_HOLD ;
1929:   ;
1930:   ;
1931:   ;
 2:  --eg:PASTE (FR50L1810) ;
1939:   ;
1940:   ;
1941:L P[589] 1000mm/sec CNT35    ;
1942:   ;
1943:J P[590] 50% CNT25    ;
1944:   ;
1945:L P[591] 1000mm/sec CNT40    ;
1946:   ;
1947:   ;
1948:  !FR50L1820 ;
1949:  IF R[15]=1822,CALL TECH_HOLD ;
1950:   ;
1951:   ;
1952:   ;
 2:  --eg:PASTE (FR50L1820) ;
1958:   ;
1959:   ;
1960:L P[595] 1000mm/sec CNT50    ;
1961:   ;
1962:J P[596] 50% CNT60    ;
1963:   ;
1964:J P[597] 50% CNT40    ;
1965:   ;
1966:L P[598] 1000mm/sec CNT25    ;
1967:   ;
1968:   ;
1969:   ;
1970:  !FR50L1830 ;
1971:  IF R[15]=1832,CALL TECH_HOLD ;
1972:   ;
1973:   ;
1974:   ;
 2:  --eg:PASTE (FR50L1830) ;
1985:   ;
1986:   ;
1987:L P[607] 1000mm/sec CNT60    ;
1988:   ;
1989:J P[608] 50% CNT50    ;
1990:   ;
1991:   ;
1992:  !FR50L1840 ;
1993:  IF R[15]=1842,CALL TECH_HOLD ;
1994:   ;
1995:   ;
1996:   ;
 2:  --eg:PASTE (FR50L1840) ;
2009:   ;
2010:   ;
2011:L P[618] 1000mm/sec CNT25    ;
2012:   ;
2013:J P[619] 50% CNT75    ;
2014:   ;
2015:J P[620] 50% CNT75    ;
2016:   ;
2017:J P[372] 50% CNT80    ;
2018:   ;
2019:L P[621] 1000mm/sec CNT40    ;
2020:   ;
2021:   ;
2022:  !FR50L1850 ;
2023:  IF R[15]=1852,CALL TECH_HOLD ;
2024:   ;
2025:   ;
 2:  --eg:PASTE (FR50L1850) ;
2032:   ;
2033:   ;
2034:L P[626] 1000mm/sec CNT90    ;
2035:   ;
2036:L P[627] 1000mm/sec CNT100    ;
2037:   ;
2038:   ;
2039:  !FR50L1860 ;
2040:  IF R[15]=1862,CALL TECH_HOLD ;
2041:   ;
2042:   ;
2043:   ;
 2:  --eg:PASTE (FR50L1860) ;
2050:   ;
2051:   ;
2052:L P[630] 1000mm/sec CNT50    ;
2053:   ;
2054:   ;
2055:  !FR50L1870 ;
2056:  IF R[15]=1872,CALL TECH_HOLD ;
2057:   ;
2058:   ;
2059:   ;
 2:  --eg:PASTE (FR50L1870) ;
2067:   ;
2068:   ;
2069:L P[634] 1000mm/sec CNT60    ;
2070:   ;
2071:   ;
2072:  !FR50L1880 ;
2073:  IF R[15]=1882,CALL TECH_HOLD ;
2074:   ;
2075:   ;
2076:   ;
 2:  --eg:PASTE (FR50L1880) ;
2084:   ;
2085:   ;
2086:L P[373] 1000mm/sec CNT25    ;
2087:   ;
2088:J P[638] 50% CNT25    ;
2089:   ;
2090:J P[641] 50% CNT25    ;
2091:   ;
2092:   ;
2093:  !FR50L1900 ;
2094:  IF R[15]=1902,CALL TECH_HOLD ;
2095:   ;
2096:   ;
2097:   ;
 2:  --eg:PASTE (FR50L1900) ;
2105:   ;
2106:   ;
2107:L P[645] 1000mm/sec CNT40    ;
2108:   ;
2109:J P[87] 50% CNT35    ;
2110:  --eg:Insert g2j2 @-90 Loadstop!!! ;
2111:   ;
2112:  !********POSITIONER MOVE******** ;
2113:J P[106] 85% CNT40    ;
2114:   ;
2115:J P[107] 50% CNT80    ;
2116:   ;
2117:   ;
2118:  !FR50L2010 ;
2119:  IF R[15]=2012,CALL TECH_HOLD ;
2120:   ;
2121:L P[108] 1000mm/sec CNT25    ;
2122:   ;
2123:   ;
 2:  --eg:PASTE (FR50L2010) ;
2133:   ;
2134:   ;
2135:  CALL ARC_LH_DISABLE_LS(1) ;
2136:   ;
2137:L P[469] 1000mm/sec CNT50    ;
2138:   ;
2139:J P[470] 50% CNT100    ;
2140:   ;
2141:J P[471] 50% CNT70    ;
2142:   ;
2143:J P[472] 50% CNT40    ;
2144:   ;
2145:  --eg:Insert g2j2 @-90 Loadstop!!! ;
2148:   ;
2149:  !********POSITIONER MOVE******** ;
2150:J P[118] 85% CNT40    ;
2151:   ;
2152:J P[646] 90% CNT50    ;
2153:   ;
2154:L P[647] 1000mm/sec CNT40    ;
2155:   ;
2156:L P[648] 1000mm/sec CNT25    ;
2157:   ;
2158:   ;
2159:  !FR50L1910 ;
2160:  IF R[15]=1912,CALL TECH_HOLD ;
2161:   ;
2162:   ;
2163:   ;
 2:  --eg:PASTE (FR50L1910) ;
2184:   ;
2185:L P[670] 1000mm/sec CNT25    ;
2186:   ;
2187:L P[671] 500mm/sec CNT25    ;
2188:   ;
2189:   ;
2190:  !FR50L1911 ;
2191:  IF R[15]=1913,CALL TECH_HOLD ;
2192:   ;
2193:   ;
 2:  --eg:PASTE (FR50L1911) ;
2203:   ;
2204:L P[679] 1000mm/sec CNT80    ;
2205:   ;
2206:L P[680] 900mm/sec CNT30 Wjnt    ;
2207:   ;
2208:J P[95] 50% CNT90    ;
2209:   ;
2210:J P[681] 50% CNT40    ;
2211:   ;
2212:  !HOME ;
2213:J P[94] 80% CNT40    ;
2214:   ;
2215:  !********POSITIONER MOVE******** ;
2216:J P[682] 90% CNT30    ;
2217:   ;
2218:J P[683] 50% CNT85    ;
2219:   ;
2220:J P[684] 50% CNT30    ;
2221:   ;
2222:L P[685] 1000mm/sec CNT25    ;
2223:   ;
2224:  !TO SKIP FRONT BUMPER WELDS ;
2225:  CALL ARC_DISABLE_FRONT_BMPR_LRG(0) ;
2226:   ;
2227:  !FR50L1920 ;
2228:  IF R[15]=1922,CALL TECH_HOLD ;
2229:   ;
2230:  UALM[20] ;
2231:  --eg:CHECK NEXT 3 WELDS ;
2232:   ;
2233:   ;
 2:  --eg:PASTE (FR50L1920) ;
2240:   ;
2241:   ;
2242:L P[688] 1000mm/sec CNT100    ;
2243:   ;
2244:J P[689] 50% CNT25    ;
2245:   ;
2246:L P[690] 1000mm/sec CNT25    ;
2247:   ;
2248:   ;
2249:  !FR50L1930 ;
2250:  IF R[15]=1932,CALL TECH_HOLD ;
2251:   ;
 2:  --eg:PASTE (FR50L1930) ;
2260:   ;
2261:   ;
2262:L P[694] 1000mm/sec CNT100    ;
2263:   ;
2264:J P[695] 16% CNT100    ;
2265:   ;
2266:  UALM[20] ;
2267:   ;
2268:  !FR50L1940 ;
2269:  IF R[15]=1942,CALL TECH_HOLD ;
2270:   ;
2271:   ;
2272:   ;
 2:  --eg:PASTE (FR50L1940) ;
2279:   ;
2280:   ;
2281:  CALL ARC_DISABLE_FRONT_BMPR_LRG(1) ;
2282:   ;
2283:L P[698] 1000mm/sec CNT25    ;
2284:   ;
2285:J P[699] 50% CNT40    ;
2286:   ;
2287:  !********POSITIONER MOVE******** ;
2288:J P[700] 90% CNT30    ;
2289:   ;
2290:J P[701] 50% CNT30    ;
2291:   ;
2292:   ;
2293:  CALL ARC_LH_DISABLE_LS(0) ;
2294:   ;
2295:  !FR50L1950 ;
2296:  IF R[15]=1952,CALL TECH_HOLD ;
2297:   ;
2298:   ;
2299:L P[702] 1000mm/sec CNT25    ;
2300:   ;
2301:   ;
 2:  --eg:PASTE (FR50L1950) ;
2310:   ;
2311:   ;
2312:  CALL ARC_LH_DISABLE_LS(1) ;
2313:   ;
2314:L P[708] 1000mm/sec CNT50    ;
2315:   ;
2316:J P[97] 50% CNT25    ;
2317:   ;
2318:J P[710] 50% CNT25    ;
2319:   ;
2320:  !********POSITIONER MOVE******** ;
2321:J P[2] 85% CNT40    ;
2322:   ;
2323:J P[105] 50% CNT25    ;
2324:   ;
2325:L P[113] 1000mm/sec CNT25    ;
2326:   ;
2327:  CALL ARC_DISABLE_RH_LS(0) ;
2328:   ;
2329:  !FR50L1970 ;
2330:  IF R[15]=1972,CALL TECH_HOLD ;
2331:   ;
2332:   ;
2333:   ;
 2:  --eg:PASTE (FR50L1970) ;
2341:   ;
2342:   ;
2343:L P[564] 800mm/sec CNT5    ;
2344:   ;
2345:J P[571] 20% CNT40    ;
2346:   ;
2347:J P[639] 40% CNT25    ;
2348:   ;
2349:J P[640] 75% CNT50    ;
2350:   ;
2351:  !********POSITIONER MOVE******** ;
2352:J P[711] 85% CNT30    ;
2353:   ;
2354:J P[712] 50% CNT80    ;
2355:   ;
2356:L P[713] 1000mm/sec CNT40    ;
2357:   ;
2358:   ;
2359:  !FR50L1960 ;
2360:  IF R[15]=1962,CALL TECH_HOLD ;
2361:   ;
2362:   ;
2363:L P[714] 500mm/sec CNT25    ;
2364:   ;
2365:   ;
 2:  --eg:PASTE (FR50L1960) ;
2374:   ;
2375:   ;
2376:  CALL ARC_DISABLE_RH_LS(1) ;
2377:   ;
2378:L P[720] 500mm/sec CNT35    ;
2379:   ;
2380:L P[721] 1000mm/sec CNT100    ;
2381:   ;
2382:J P[99] 100% CNT30    ;
2383:   ;
2384:  !******** POSITIONER MOVE ******* ;
2385:J P[793] 85% CNT30    ;
2386:   ;
2387:J P[732] 75% CNT25    ;
2388:   ;
2389:L P[733] 1000mm/sec CNT100    ;
2390:   ;
2391:   ;
2392:  CALL ARC_LH_DISABLE_LS(0) ;
2393:   ;
2394:  !FR50L1980 ;
2395:  IF R[15]=1982,CALL TECH_HOLD ;
2396:   ;
2397:   ;
2398:   ;
 2:  --eg:PASTE (FR50L1980) ;
2406:   ;
2407:   ;
2408:L P[738] 800mm/sec CNT20    ;
2409:   ;
2410:L P[739] 1000mm/sec CNT100    ;
2411:   ;
2412:J P[740] 100% CNT100    ;
2413:   ;
2414:  !HOME ;
2415:J P[104] 100% CNT30    ;
2416:   ;
2417:  CALL HOME    ;
2418:   ;
2419:  !********POSITIONER MOVE******** ;
2420:  CALL LOAD_POS    ;
2421:   ;
2422:  R[79:TEST LRG WELDDIT]=($AWEPRODSTAT[1].$WELD_DIST) ;
/POS
P[1]{
   GP1:
	UF : 1, UT : 1,		CONFIG : 'N U T, 0, 0, 0',
	X =  1048.285  mm,	Y = -1294.070  mm,	Z =   701.250  mm,
	W =     -.009 deg,	P =    41.863 deg,	R =  -150.867 deg
   GP2:
	UF : 1, UT : 1,
	J1=     0.000 deg,	J2=   -40.000 deg
};
P[2]{
   GP1:
	UF : 1, UT : 1,		CONFIG : 'N U T, 0, 0, 0',
	X =  1171.584  mm,	Y = -1326.619  mm,	Z =  1560.411  mm,
	W =   -31.995 deg,	P =   -11.977 deg,	R =    17.020 deg
   GP2:
	UF : 1, UT : 1,
	J1=   180.000 deg,	J2=  -125.000 deg
};
P[3]{
   GP1:
	UF : 1, UT : 1,		CONFIG : 'N U T, 0, 0, 0',
	X =  1209.555  mm,	Y = -1322.972  mm,	Z =   229.179  mm,
	W =     -.010 deg,	P =    41.970 deg,	R =  -145.526 deg
   GP2:
	UF : 1, UT : 1,
	J1=     0.000 deg,	J2=   -40.000 deg
};
P[4]{
   GP1:
	UF : 1, UT : 1,		CONFIG : 'N U B, 0, 0, 0',
	X =   356.032  mm,	Y =    -2.146  mm,	Z =  2424.050  mm,
	W =      .001 deg,	P =   -40.002 deg,	R =     -.005 deg
   GP2:
	UF : 1, UT : 1,
	J1=     0.000 deg,	J2=   -40.000 deg
};
P[5]{
   GP1:
	UF : 1, UT : 1,		CONFIG : 'N U T, 0, 0, 0',
	X =  1247.331  mm,	Y = -1259.850  mm,	Z =    76.111  mm,
	W =    -2.552 deg,	P =    43.819 deg,	R =  -145.577 deg
   GP2:
	UF : 1, UT : 1,
	J1=     0.000 deg,	J2=   -40.000 deg
};
P[6]{
   GP1:
	UF : 1, UT : 1,		CONFIG : 'N U T, 0, 0, 0',
	X =  1293.538  mm,	Y = -1316.451  mm,	Z =    78.580  mm,
	W =    -2.838 deg,	P =    43.807 deg,	R =  -171.689 deg
   GP2:
	UF : 1, UT : 1,
	J1=     0.000 deg,	J2=   -40.000 deg
};
P[7]{
   GP1:
	UF : 1, UT : 1,		CONFIG : 'N U B, 0, 0, 0',
	X =   356.032  mm,	Y =    -2.146  mm,	Z =  2424.049  mm,
	W =      .001 deg,	P =   -40.002 deg,	R =     -.005 deg
   GP2:
	UF : 1, UT : 1,
	J1=    45.000 deg,	J2=     0.000 deg
};
P[8]{
   GP1:
	UF : 1, UT : 1,		CONFIG : 'N U T, 0, 0, 0',
	X =  1272.049  mm,	Y = -1319.952  mm,	Z =   170.275  mm,
	W =    -4.003 deg,	P =    44.859 deg,	R =  -166.486 deg
   GP2:
	UF : 1, UT : 1,
	J1=     0.000 deg,	J2=   -40.000 deg
};
P[9]{
   GP1:
	UF : 1, UT : 1,		CONFIG : 'N U T, 0, 0, 0',
	X =   909.960  mm,	Y =  -872.839  mm,	Z =   170.274  mm,
	W =      .297 deg,	P =    44.999 deg,	R =  -138.174 deg
   GP2:
	UF : 1, UT : 1,
	J1=     0.000 deg,	J2=   -40.000 deg
};
P[10]{
   GP1:
	UF : 1, UT : 1,		CONFIG : 'N U T, 0, 0, 0',
	X =   887.983  mm,	Y =  -832.584  mm,	Z =    82.605  mm,
	W =      .290 deg,	P =    45.004 deg,	R =  -138.180 deg
   GP2:
	UF : 1, UT : 1,
	J1=     0.000 deg,	J2=   -40.000 deg
};
P[11]{
   GP1:
	UF : 1, UT : 1,		CONFIG : 'N U T, 0, 0, 0',
	X =  1224.457  mm,	Y = -1231.721  mm,	Z =    74.809  mm,
	W =      .871 deg,	P =    43.917 deg,	R =  -137.698 deg
   GP2:
	UF : 1, UT : 1,
	J1=     0.000 deg,	J2=   -40.000 deg
};
P[12]{
   GP1:
	UF : 1, UT : 1,		CONFIG : 'N U T, 0, 0, 0',
	X =  1163.391  mm,	Y = -1298.112  mm,	Z =   230.228  mm,
	W =     1.291 deg,	P =    44.986 deg,	R =  -138.174 deg
   GP2:
	UF : 1, UT : 1,
	J1=     0.000 deg,	J2=   -40.000 deg
};
P[13]{
   GP1:
	UF : 1, UT : 1,		CONFIG : 'N U T, 0, 0, 0',
	X =   860.828  mm,	Y =  -857.112  mm,	Z =   230.228  mm,
	W =     1.291 deg,	P =    44.986 deg,	R =  -138.174 deg
   GP2:
	UF : 1, UT : 1,
	J1=     0.000 deg,	J2=   -40.000 deg
};
P[14]{
   GP1:
	UF : 1, UT : 1,		CONFIG : 'N U T, 0, 0, 0',
	X =   865.839  mm,	Y =  -805.519  mm,	Z =    81.655  mm,
	W =     1.287 deg,	P =    44.985 deg,	R =  -138.181 deg
   GP2:
	UF : 1, UT : 1,
	J1=     0.000 deg,	J2=   -40.000 deg
};
P[15]{
   GP1:
	UF : 1, UT : 1,		CONFIG : 'N U T, 0, 0, 0',
	X =   820.424  mm,	Y =  -752.765  mm,	Z =    81.650  mm,
	W =     1.452 deg,	P =    44.761 deg,	R =  -108.453 deg
   GP2:
	UF : 1, UT : 1,
	J1=     0.000 deg,	J2=   -40.000 deg
};
P[16]{
   GP1:
	UF : 1, UT : 1,		CONFIG : 'N U T, 0, 0, 0',
	X =   643.854  mm,	Y = -1045.560  mm,	Z =   456.782  mm,
	W =     1.290 deg,	P =    44.986 deg,	R =  -124.491 deg
   GP2:
	UF : 1, UT : 1,
	J1=     0.000 deg,	J2=   -40.000 deg
};
P[17]{
   GP1:
	UF : 1, UT : 1,		CONFIG : 'N U T, 0, 0, 0',
	X =   908.243  mm,	Y =     -.972  mm,	Z =  2177.323  mm,
	W =     -.010 deg,	P =   -45.000 deg,	R =     0.000 deg
   GP2:
	UF : 1, UT : 1,
	J1=    90.000 deg,	J2=     0.000 deg
};
P[18]{
   GP1:
	UF : 1, UT : 1,		CONFIG : 'N U T, 0, 0, 0',
	X =  1593.884  mm,	Y =    54.651  mm,	Z =  1425.564  mm,
	W =    40.560 deg,	P =     2.984 deg,	R =   -28.829 deg
   GP2:
	UF : 1, UT : 1,
	J1=    90.000 deg,	J2=     0.000 deg
};
P[19]{
   GP1:
	UF : 1, UT : 1,		CONFIG : 'N U T, 0, 0, 0',
	X =  2419.244  mm,	Y =   170.457  mm,	Z =   756.322  mm,
	W =    40.554 deg,	P =     2.977 deg,	R =   -28.823 deg
   GP2:
	UF : 1, UT : 1,
	J1=    90.000 deg,	J2=     0.000 deg
};
P[20]{
   GP1:
	UF : 1, UT : 1,		CONFIG : 'N U T, 0, 0, 0',
	X =  2486.244  mm,	Y =   320.457  mm,	Z =   579.520  mm,
	W =    40.554 deg,	P =     2.977 deg,	R =    -7.352 deg
   GP2:
	UF : 1, UT : 1,
	J1=    90.000 deg,	J2=     0.000 deg
};
P[21]{
   GP1:
	UF : 1, UT : 1,		CONFIG : 'N U T, 0, 0, 0',
	X =  2501.284  mm,	Y =   410.619  mm,	Z =   482.746  mm,
	W =    44.788 deg,	P =     5.020 deg,	R =    -1.194 deg
   GP2:
	UF : 1, UT : 1,
	J1=    90.000 deg,	J2=     0.000 deg
};
P[22]{
   GP1:
	UF : 1, UT : 1,		CONFIG : 'N U T, 0, 0, 0',
	X =  2460.572  mm,	Y =   411.691  mm,	Z =   482.746  mm,
	W =    44.788 deg,	P =     5.020 deg,	R =    -1.194 deg
   GP2:
	UF : 1, UT : 1,
	J1=    90.000 deg,	J2=     0.000 deg
};
P[23]{
   GP1:
	UF : 1, UT : 1,		CONFIG : 'N U T, 0, 0, 0',
	X =  2439.697  mm,	Y =   412.351  mm,	Z =   484.565  mm,
	W =    44.788 deg,	P =     5.020 deg,	R =    30.332 deg
   GP2:
	UF : 1, UT : 1,
	J1=    90.000 deg,	J2=     0.000 deg
};
P[24]{
   GP1:
	UF : 1, UT : 1,		CONFIG : 'N U T, 0, 0, 0',
	X =  2521.819  mm,	Y =   261.320  mm,	Z =   656.993  mm,
	W =    44.759 deg,	P =     5.240 deg,	R =    21.047 deg
   GP2:
	UF : 1, UT : 1,
	J1=    90.000 deg,	J2=     0.000 deg
};
P[25]{
   GP1:
	UF : 1, UT : 1,		CONFIG : 'N U T, 0, 0, 0',
	X =  2511.367  mm,	Y =  -251.873  mm,	Z =   577.119  mm,
	W =   -39.345 deg,	P =     9.413 deg,	R =    11.283 deg
   GP2:
	UF : 1, UT : 1,
	J1=    90.000 deg,	J2=     0.000 deg
};
P[26]{
   GP1:
	UF : 1, UT : 1,		CONFIG : 'N U T, 0, 0, 0',
	X =  2521.216  mm,	Y =  -413.066  mm,	Z =   490.603  mm,
	W =   -44.053 deg,	P =    10.305 deg,	R =     9.161 deg
   GP2:
	UF : 1, UT : 1,
	J1=    90.000 deg,	J2=     0.000 deg
};
P[27]{
   GP1:
	UF : 1, UT : 1,		CONFIG : 'N U T, 0, 0, 0',
	X =  2473.788  mm,	Y =  -413.066  mm,	Z =   490.604  mm,
	W =   -44.053 deg,	P =    10.305 deg,	R =     9.161 deg
   GP2:
	UF : 1, UT : 1,
	J1=    90.000 deg,	J2=     0.000 deg
};
P[28]{
   GP1:
	UF : 1, UT : 1,		CONFIG : 'N U T, 0, 0, 0',
	X =  2447.042  mm,	Y =  -413.341  mm,	Z =   492.423  mm,
	W =   -44.053 deg,	P =    10.305 deg,	R =   -18.834 deg
   GP2:
	UF : 1, UT : 1,
	J1=    90.000 deg,	J2=     0.000 deg
};
P[29]{
   GP1:
	UF : 1, UT : 1,		CONFIG : 'N U T, 0, 0, 0',
	X =  2549.787  mm,	Y =  -262.671  mm,	Z =   682.477  mm,
	W =   -44.052 deg,	P =    10.305 deg,	R =   -20.066 deg
   GP2:
	UF : 1, UT : 1,
	J1=    90.000 deg,	J2=     0.000 deg
};
P[30]{
   GP1:
	UF : 1, UT : 1,		CONFIG : 'N U T, 0, 0, 0',
	X =  2103.073  mm,	Y =   282.472  mm,	Z =   462.977  mm,
	W =    30.589 deg,	P =    34.770 deg,	R =    43.796 deg
   GP2:
	UF : 1, UT : 1,
	J1=    90.000 deg,	J2=     0.000 deg
};
P[31]{
   GP1:
	UF : 1, UT : 1,		CONFIG : 'N U T, 0, 0, 0',
	X =  2006.585  mm,	Y =   396.692  mm,	Z =   354.220  mm,
	W =    43.291 deg,	P =    13.764 deg,	R =    75.822 deg
   GP2:
	UF : 1, UT : 1,
	J1=    90.000 deg,	J2=     0.000 deg
};
P[32]{
   GP1:
	UF : 1, UT : 1,		CONFIG : 'N U T, 0, 0, 0',
	X =  2003.822  mm,	Y =   315.992  mm,	Z =   352.006  mm,
	W =    43.281 deg,	P =    13.759 deg,	R =    75.826 deg
   GP2:
	UF : 1, UT : 1,
	J1=    90.000 deg,	J2=     0.000 deg
};
P[33]{
   GP1:
	UF : 1, UT : 1,		CONFIG : 'N U T, 0, 0, 0',
	X =  2084.488  mm,	Y =   314.464  mm,	Z =   441.765  mm,
	W =    43.281 deg,	P =    13.759 deg,	R =    75.826 deg
   GP2:
	UF : 1, UT : 1,
	J1=    90.000 deg,	J2=     0.000 deg
};
P[34]{
   GP1:
	UF : 1, UT : 1,		CONFIG : 'N U T, 0, 0, 0',
	X =  2086.988  mm,	Y =  -331.633  mm,	Z =   441.764  mm,
	W =   -41.228 deg,	P =    19.917 deg,	R =   -68.756 deg
   GP2:
	UF : 1, UT : 1,
	J1=    90.000 deg,	J2=     0.000 deg
};
P[35]{
   GP1:
	UF : 1, UT : 1,		CONFIG : 'N U T, 0, 0, 0',
	X =  2005.569  mm,	Y =  -400.083  mm,	Z =   355.996  mm,
	W =   -41.229 deg,	P =    19.917 deg,	R =   -68.757 deg
   GP2:
	UF : 1, UT : 1,
	J1=    90.000 deg,	J2=     0.000 deg
};
P[36]{
   GP1:
	UF : 1, UT : 1,		CONFIG : 'N U T, 0, 0, 0',
	X =  2005.354  mm,	Y =  -319.297  mm,	Z =   355.996  mm,
	W =   -41.229 deg,	P =    19.917 deg,	R =   -68.757 deg
   GP2:
	UF : 1, UT : 1,
	J1=    90.000 deg,	J2=     0.000 deg
};
P[37]{
   GP1:
	UF : 1, UT : 1,		CONFIG : 'N U T, 0, 0, 0',
	X =  2106.807  mm,	Y =  -322.474  mm,	Z =   465.914  mm,
	W =   -41.228 deg,	P =    19.917 deg,	R =   -68.756 deg
   GP2:
	UF : 1, UT : 1,
	J1=    90.000 deg,	J2=     0.000 deg
};
P[38]{
   GP1:
	UF : 1, UT : 1,		CONFIG : 'N U T, 0, 0, 0',
	X =  2109.307  mm,	Y =    75.081  mm,	Z =   465.913  mm,
	W =     3.207 deg,	P =    44.910 deg,	R =   -85.462 deg
   GP2:
	UF : 1, UT : 1,
	J1=    90.000 deg,	J2=     0.000 deg
};
P[39]{
   GP1:
	UF : 1, UT : 1,		CONFIG : 'N U T, 0, 0, 0',
	X =  2681.306  mm,	Y =  -103.919  mm,	Z =  -438.087  mm,
	W =    -1.257 deg,	P =    33.277 deg,	R =   -88.589 deg
   GP2:
	UF : 1, UT : 1,
	J1=    90.000 deg,	J2=     0.000 deg
};
P[40]{
   GP1:
	UF : 1, UT : 1,		CONFIG : 'N U T, 0, 0, 0',
	X =  2726.810  mm,	Y =   -59.880  mm,	Z =  -600.102  mm,
	W =      .970 deg,	P =    44.992 deg,	R =   -88.627 deg
   GP2:
	UF : 1, UT : 1,
	J1=    90.000 deg,	J2=     0.000 deg
};
P[41]{
   GP1:
	UF : 1, UT : 1,		CONFIG : 'N U T, 0, 0, 0',
	X =  2756.313  mm,	Y =   -62.356  mm,	Z =  -598.555  mm,
	W =      .970 deg,	P =    44.992 deg,	R =   -88.627 deg
   GP2:
	UF : 1, UT : 1,
	J1=    90.000 deg,	J2=     0.000 deg
};
P[42]{
   GP1:
	UF : 1, UT : 1,		CONFIG : 'N U T, 0, 0, 0',
	X =  2676.306  mm,	Y =  -106.919  mm,	Z =  -439.087  mm,
	W =    -1.257 deg,	P =    33.277 deg,	R =   -88.589 deg
   GP2:
	UF : 1, UT : 1,
	J1=    90.000 deg,	J2=     0.000 deg
};
P[43]{
   GP1:
	UF : 1, UT : 1,		CONFIG : 'N U T, 0, 0, 0',
	X =  2576.306  mm,	Y =    -6.919  mm,	Z =  -439.087  mm,
	W =    -1.257 deg,	P =    33.277 deg,	R =   -88.589 deg
   GP2:
	UF : 1, UT : 1,
	J1=    90.000 deg,	J2=     0.000 deg
};
P[44]{
   GP1:
	UF : 1, UT : 1,		CONFIG : 'N U T, 0, 0, 0',
	X =  2582.224  mm,	Y =   118.706  mm,	Z =  -400.809  mm,
	W =      .677 deg,	P =    39.803 deg,	R =    91.170 deg
   GP2:
	UF : 1, UT : 1,
	J1=    90.000 deg,	J2=     0.000 deg
};
P[45]{
   GP1:
	UF : 1, UT : 1,		CONFIG : 'N U T, 0, 0, 0',
	X =  2706.224  mm,	Y =   118.706  mm,	Z =  -483.809  mm,
	W =      .677 deg,	P =    39.803 deg,	R =    91.170 deg
   GP2:
	UF : 1, UT : 1,
	J1=    90.000 deg,	J2=     0.000 deg
};
P[46]{
   GP1:
	UF : 1, UT : 1,		CONFIG : 'N U T, 0, 0, 0',
	X =  2726.713  mm,	Y =    53.817  mm,	Z =  -600.251  mm,
	W =      .895 deg,	P =    44.993 deg,	R =    91.267 deg
   GP2:
	UF : 1, UT : 1,
	J1=    90.000 deg,	J2=     0.000 deg
};
P[47]{
   GP1:
	UF : 1, UT : 1,		CONFIG : 'N U T, 0, 0, 0',
	X =  2754.017  mm,	Y =    54.236  mm,	Z =  -600.074  mm,
	W =      .893 deg,	P =    44.993 deg,	R =    91.262 deg
   GP2:
	UF : 1, UT : 1,
	J1=    90.000 deg,	J2=     0.000 deg
};
P[48]{
   GP1:
	UF : 1, UT : 1,		CONFIG : 'N U T, 0, 0, 0',
	X =  2706.224  mm,	Y =   118.706  mm,	Z =  -483.809  mm,
	W =      .677 deg,	P =    39.803 deg,	R =    91.170 deg
   GP2:
	UF : 1, UT : 1,
	J1=    90.000 deg,	J2=     0.000 deg
};
P[49]{
   GP1:
	UF : 1, UT : 1,		CONFIG : 'N U T, 0, 0, 0',
	X =  2750.938  mm,	Y =   112.285  mm,	Z =  -474.250  mm,
	W =     -.713 deg,	P =    25.922 deg,	R =     -.241 deg
   GP2:
	UF : 1, UT : 1,
	J1=    90.000 deg,	J2=     0.000 deg
};
P[50]{
   GP1:
	UF : 1, UT : 1,		CONFIG : 'N U T, 0, 0, 0',
	X =  2778.081  mm,	Y =    53.285  mm,	Z =  -487.998  mm,
	W =     -.713 deg,	P =    25.922 deg,	R =     -.241 deg
   GP2:
	UF : 1, UT : 1,
	J1=    90.000 deg,	J2=     0.000 deg
};
P[51]{
   GP1:
	UF : 1, UT : 1,		CONFIG : 'N U T, 0, 0, 0',
	X =  2760.865  mm,	Y =    49.400  mm,	Z =  -601.908  mm,
	W =     -.646 deg,	P =    35.845 deg,	R =     -.312 deg
   GP2:
	UF : 1, UT : 1,
	J1=    89.996 deg,	J2=     0.000 deg
};
P[52]{
   GP1:
	UF : 1, UT : 1,		CONFIG : 'N U T, 0, 0, 0',
	X =  2760.669  mm,	Y =   -52.646  mm,	Z =  -601.987  mm,
	W =     -.641 deg,	P =    35.842 deg,	R =     -.313 deg
   GP2:
	UF : 1, UT : 1,
	J1=    89.996 deg,	J2=     0.000 deg
};
P[53]{
   GP1:
	UF : 1, UT : 1,		CONFIG : 'N U T, 0, 0, 0',
	X =  2774.367  mm,	Y =   -45.046  mm,	Z =  -326.584  mm,
	W =     -.063 deg,	P =     6.406 deg,	R =     -.319 deg
   GP2:
	UF : 1, UT : 1,
	J1=    90.000 deg,	J2=     0.000 deg
};
P[54]{
   GP1:
	UF : 1, UT : 1,		CONFIG : 'N U T, 0, 0, 0',
	X =  2318.510  mm,	Y =     4.126  mm,	Z =   836.416  mm,
	W =     -.063 deg,	P =     6.406 deg,	R =     -.319 deg
   GP2:
	UF : 1, UT : 1,
	J1=    90.000 deg,	J2=     0.000 deg
};
P[55]{
   GP1:
	UF : 1, UT : 1,		CONFIG : 'N U T, 0, 0, 0',
	X =  2651.064  mm,	Y =   274.146  mm,	Z =   596.222  mm,
	W =    40.438 deg,	P =    -1.956 deg,	R =     2.337 deg
   GP2:
	UF : 1, UT : 1,
	J1=    90.000 deg,	J2=     0.000 deg
};
P[56]{
   GP1:
	UF : 1, UT : 1,		CONFIG : 'N U T, 0, 0, 0',
	X =  2678.366  mm,	Y =   323.391  mm,	Z =   552.416  mm,
	W =    40.027 deg,	P =    -6.599 deg,	R =     7.835 deg
   GP2:
	UF : 1, UT : 1,
	J1=    90.000 deg,	J2=     0.000 deg
};
P[57]{
   GP1:
	UF : 1, UT : 1,		CONFIG : 'N U T, 0, 0, 0',
	X =  2754.430  mm,	Y =   412.446  mm,	Z =   451.473  mm,
	W =    44.541 deg,	P =    -7.214 deg,	R =     7.272 deg
   GP2:
	UF : 1, UT : 1,
	J1=    90.000 deg,	J2=     0.000 deg
};
P[58]{
   GP1:
	UF : 1, UT : 1,		CONFIG : 'N U T, 0, 0, 0',
	X =  2707.644  mm,	Y =   412.446  mm,	Z =   451.473  mm,
	W =    44.541 deg,	P =    -7.214 deg,	R =     7.272 deg
   GP2:
	UF : 1, UT : 1,
	J1=    90.000 deg,	J2=     0.000 deg
};
P[59]{
   GP1:
	UF : 1, UT : 1,		CONFIG : 'N U T, 0, 0, 0',
	X =  2698.437  mm,	Y =   269.508  mm,	Z =   599.906  mm,
	W =    44.541 deg,	P =    -7.214 deg,	R =     7.272 deg
   GP2:
	UF : 1, UT : 1,
	J1=    90.000 deg,	J2=     0.000 deg
};
P[60]{
   GP1:
	UF : 1, UT : 1,		CONFIG : 'N U T, 0, 0, 0',
	X =  2703.937  mm,	Y =  -282.492  mm,	Z =   602.906  mm,
	W =   -34.404 deg,	P =     5.822 deg,	R =     8.425 deg
   GP2:
	UF : 1, UT : 1,
	J1=    90.000 deg,	J2=     0.000 deg
};
P[61]{
   GP1:
	UF : 1, UT : 1,		CONFIG : 'N U T, 0, 0, 0',
	X =  2753.662  mm,	Y =  -414.958  mm,	Z =   454.284  mm,
	W =   -44.541 deg,	P =     7.214 deg,	R =     7.272 deg
   GP2:
	UF : 1, UT : 1,
	J1=    90.000 deg,	J2=     0.000 deg
};
P[62]{
   GP1:
	UF : 1, UT : 1,		CONFIG : 'N U T, 0, 0, 0',
	X =  2708.519  mm,	Y =  -415.387  mm,	Z =   454.284  mm,
	W =   -44.541 deg,	P =     7.214 deg,	R =     7.272 deg
   GP2:
	UF : 1, UT : 1,
	J1=    90.000 deg,	J2=     0.000 deg
};
P[63]{
   GP1:
	UF : 1, UT : 1,		CONFIG : 'N U T, 0, 0, 0',
	X =  2699.988  mm,	Y =  -282.600  mm,	Z =   597.231  mm,
	W =   -44.541 deg,	P =     7.214 deg,	R =     7.272 deg
   GP2:
	UF : 1, UT : 1,
	J1=    90.000 deg,	J2=     0.000 deg
};
P[64]{
   GP1:
	UF : 1, UT : 1,		CONFIG : 'F U T, 0, 0, 0',
	X =  2542.011  mm,	Y =    62.997  mm,	Z =   733.500  mm,
	W =      .337 deg,	P =   -50.731 deg,	R =     6.061 deg
   GP2:
	UF : 1, UT : 1,
	J1=    90.000 deg,	J2=     0.000 deg
};
P[65]{
   GP1:
	UF : 1, UT : 1,		CONFIG : 'F U T, 0, 0, 0',
	X =  2864.014  mm,	Y =   282.441  mm,	Z =   502.065  mm,
	W =   -15.171 deg,	P =   -43.175 deg,	R =    33.524 deg
   GP2:
	UF : 1, UT : 1,
	J1=    90.000 deg,	J2=     0.000 deg
};
P[66]{
   GP1:
	UF : 1, UT : 1,		CONFIG : 'F U T, 0, 0, 0',
	X =  2900.162  mm,	Y =   279.864  mm,	Z =   453.527  mm,
	W =   -15.171 deg,	P =   -43.175 deg,	R =    33.523 deg
   GP2:
	UF : 1, UT : 1,
	J1=    90.000 deg,	J2=     0.000 deg
};
P[67]{
   GP1:
	UF : 1, UT : 1,		CONFIG : 'F U T, 0, 0, 0',
	X =  2899.731  mm,	Y =   375.578  mm,	Z =   453.525  mm,
	W =    -8.441 deg,	P =   -43.927 deg,	R =    33.763 deg
   GP2:
	UF : 1, UT : 1,
	J1=    90.000 deg,	J2=     0.000 deg
};
P[68]{
   GP1:
	UF : 1, UT : 1,		CONFIG : 'F U T, 0, 0, 0',
	X =  2899.731  mm,	Y =   395.863  mm,	Z =   453.523  mm,
	W =    -2.617 deg,	P =   -43.940 deg,	R =    39.916 deg
   GP2:
	UF : 1, UT : 1,
	J1=    90.000 deg,	J2=     0.000 deg
};
P[69]{
   GP1:
	UF : 1, UT : 1,		CONFIG : 'F U T, 0, 0, 0',
	X =  2894.517  mm,	Y =   408.077  mm,	Z =   453.523  mm,
	W =    -2.617 deg,	P =   -43.939 deg,	R =    53.826 deg
   GP2:
	UF : 1, UT : 1,
	J1=    90.000 deg,	J2=     0.000 deg
};
P[70]{
   GP1:
	UF : 1, UT : 1,		CONFIG : 'F U T, 0, 0, 0',
	X =  2879.587  mm,	Y =   413.648  mm,	Z =   453.520  mm,
	W =    -2.617 deg,	P =   -43.939 deg,	R =    78.094 deg
   GP2:
	UF : 1, UT : 1,
	J1=    90.000 deg,	J2=     0.000 deg
};
P[71]{
   GP1:
	UF : 1, UT : 1,		CONFIG : 'F U T, 0, 0, 0',
	X =  2876.300  mm,	Y =   413.648  mm,	Z =   453.519  mm,
	W =    -2.617 deg,	P =   -43.939 deg,	R =    78.094 deg
   GP2:
	UF : 1, UT : 1,
	J1=    90.000 deg,	J2=     0.000 deg
};
P[72]{
   GP1:
	UF : 1, UT : 1,		CONFIG : 'F U T, 0, 0, 0',
	X =  2697.000  mm,	Y =   247.797  mm,	Z =   648.652  mm,
	W =    -2.629 deg,	P =   -43.936 deg,	R =    42.269 deg
   GP2:
	UF : 1, UT : 1,
	J1=    90.000 deg,	J2=     0.000 deg
};
P[73]{
   GP1:
	UF : 1, UT : 1,		CONFIG : 'N U T, 0, 0, 0',
	X =   949.898  mm,	Y =    98.916  mm,	Z =  1480.357  mm,
	W =   -25.667 deg,	P =   -34.352 deg,	R =    34.753 deg
   GP2:
	UF : 1, UT : 1,
	J1=     0.000 deg,	J2=   180.000 deg
};
P[74]{
   GP1:
	UF : 1, UT : 1,		CONFIG : 'N U T, 1, 0, 0',
	X =  2528.555  mm,	Y =   -65.615  mm,	Z =   892.718  mm,
	W =   -11.578 deg,	P =   -57.733 deg,	R =     8.895 deg
   GP2:
	UF : 1, UT : 1,
	J1=    90.000 deg,	J2=     0.000 deg
};
P[75]{
   GP1:
	UF : 1, UT : 1,		CONFIG : 'N U T, 0, 0, 0',
	X =  2860.056  mm,	Y =  -309.345  mm,	Z =   520.586  mm,
	W =    14.883 deg,	P =   -42.517 deg,	R =   -27.206 deg
   GP2:
	UF : 1, UT : 1,
	J1=    90.000 deg,	J2=     0.000 deg
};
P[76]{
   GP1:
	UF : 1, UT : 1,		CONFIG : 'N U T, 0, 0, 0',
	X =  2900.184  mm,	Y =  -282.896  mm,	Z =   454.158  mm,
	W =    14.883 deg,	P =   -42.517 deg,	R =   -27.206 deg
   GP2:
	UF : 1, UT : 1,
	J1=    90.000 deg,	J2=     0.000 deg
};
P[77]{
   GP1:
	UF : 1, UT : 1,		CONFIG : 'N U T, 0, 0, 0',
	X =  2900.185  mm,	Y =  -377.396  mm,	Z =   454.156  mm,
	W =     7.397 deg,	P =   -43.869 deg,	R =   -27.794 deg
   GP2:
	UF : 1, UT : 1,
	J1=    90.000 deg,	J2=     0.000 deg
};
P[78]{
   GP1:
	UF : 1, UT : 1,		CONFIG : 'N U T, 0, 0, 0',
	X =  2899.756  mm,	Y =  -400.539  mm,	Z =   454.157  mm,
	W =     7.397 deg,	P =   -43.869 deg,	R =   -33.010 deg
   GP2:
	UF : 1, UT : 1,
	J1=    90.000 deg,	J2=     0.000 deg
};
P[79]{
   GP1:
	UF : 1, UT : 1,		CONFIG : 'N U T, 0, 0, 0',
	X =  2893.399  mm,	Y =  -411.682  mm,	Z =   454.157  mm,
	W =     1.613 deg,	P =   -43.869 deg,	R =   -48.206 deg
   GP2:
	UF : 1, UT : 1,
	J1=    90.000 deg,	J2=     0.000 deg
};
P[80]{
   GP1:
	UF : 1, UT : 1,		CONFIG : 'N U T, 0, 0, 0',
	X =  2881.970  mm,	Y =  -415.825  mm,	Z =   454.156  mm,
	W =     1.613 deg,	P =   -43.869 deg,	R =   -74.666 deg
   GP2:
	UF : 1, UT : 1,
	J1=    90.000 deg,	J2=     0.000 deg
};
P[81]{
   GP1:
	UF : 1, UT : 1,		CONFIG : 'N U T, 0, 0, 0',
	X =  2874.898  mm,	Y =  -416.681  mm,	Z =   454.155  mm,
	W =     1.613 deg,	P =   -43.869 deg,	R =   -76.087 deg
   GP2:
	UF : 1, UT : 1,
	J1=    90.000 deg,	J2=     0.000 deg
};
P[82]{
   GP1:
	UF : 1, UT : 1,		CONFIG : 'N U T, 0, 0, 0',
	X =  2690.549  mm,	Y =  -310.856  mm,	Z =   600.282  mm,
	W =     1.613 deg,	P =   -43.868 deg,	R =   -40.404 deg
   GP2:
	UF : 1, UT : 1,
	J1=    90.000 deg,	J2=     0.000 deg
};
P[83]{
   GP1:
	UF : 1, UT : 1,		CONFIG : 'F U T, 0, 0, 0',
	X =  2542.011  mm,	Y =    62.997  mm,	Z =   733.500  mm,
	W =      .337 deg,	P =   -50.731 deg,	R =     6.061 deg
   GP2:
	UF : 1, UT : 1,
	J1=    90.000 deg,	J2=     0.000 deg
};
P[84]{
   GP1:
	UF : 1, UT : 1,		CONFIG : 'F U T, 0, 0, 0',
	X =  2864.014  mm,	Y =   282.441  mm,	Z =   502.065  mm,
	W =   -15.171 deg,	P =   -43.175 deg,	R =    33.524 deg
   GP2:
	UF : 1, UT : 1,
	J1=    90.000 deg,	J2=     0.000 deg
};
P[85]{
   GP1:
	UF : 1, UT : 1,		CONFIG : 'N U T, 0, 0, 0',
	X =  2172.059  mm,	Y =  -149.810  mm,	Z =  -336.475  mm,
	W =    -4.848 deg,	P =     4.640 deg,	R =    10.727 deg
   GP2:
	UF : 1, UT : 1,
	J1=    45.000 deg,	J2=   182.246 deg
};
P[86]{
   GP1:
	UF : 1, UT : 1,		CONFIG : 'N U T, 0, 0, 0',
	X =  1780.474  mm,	Y =    29.584  mm,	Z =   -67.946  mm,
	W =    -4.424 deg,	P =     7.600 deg,	R =    11.037 deg
   GP2:
	UF : 1, UT : 1,
	J1=    45.000 deg,	J2=   182.246 deg
};
P[87]{
   GP1:
	UF : 1, UT : 1,		CONFIG : 'N U T, 0, 0, 0',
	X =  1142.160  mm,	Y =  -217.183  mm,	Z =   141.822  mm,
	W =    36.993 deg,	P =    27.706 deg,	R =  -162.803 deg
   GP2:
	UF : 1, UT : 1,
	J1=    90.000 deg,	J2=   -90.000 deg
};
P[88]{
   GP1:
	UF : 1, UT : 1,		CONFIG : 'N U T, 0, 0, 0',
	X =  1987.244  mm,	Y =     -.972  mm,	Z =  1525.322  mm,
	W =     -.010 deg,	P =    45.000 deg,	R =    90.000 deg
   GP2:
	UF : 1, UT : 1,
	J1=    90.000 deg,	J2=    90.000 deg
};
P[89]{
   GP1:
	UF : 1, UT : 1,		CONFIG : 'N U T, 0, 0, 0',
	X =  2298.943  mm,	Y =    15.028  mm,	Z =   995.580  mm,
	W =   -33.416 deg,	P =    -1.271 deg,	R =    34.407 deg
   GP2:
	UF : 1, UT : 1,
	J1=    89.999 deg,	J2=   -90.000 deg
};
P[90]{
   GP1:
	UF : 1, UT : 1,		CONFIG : 'N U T, 0, 0, 0',
	X =  2543.411  mm,	Y =   825.451  mm,	Z =   -76.912  mm,
	W =   -31.199 deg,	P =     9.620 deg,	R =   105.426 deg
   GP2:
	UF : 1, UT : 1,
	J1=    80.000 deg,	J2=   -90.000 deg
};
P[91]{
   GP1:
	UF : 1, UT : 1,		CONFIG : 'F U T, 0, 0, 0',
	X =  2701.500  mm,	Y =   248.797  mm,	Z =   650.852  mm,
	W =    -2.629 deg,	P =   -43.936 deg,	R =    42.269 deg
   GP2:
	UF : 1, UT : 1,
	J1=    90.000 deg,	J2=     0.000 deg
};
P[92]{
   GP1:
	UF : 1, UT : 1,		CONFIG : 'F U T, 0, 0, 0',
	X =  2542.011  mm,	Y =    62.997  mm,	Z =   733.500  mm,
	W =      .337 deg,	P =   -50.731 deg,	R =     6.061 deg
   GP2:
	UF : 1, UT : 1,
	J1=    90.000 deg,	J2=     0.000 deg
};
P[93]{
   GP1:
	UF : 1, UT : 1,		CONFIG : 'F U T, 0, 0, 0',
	X =  2864.014  mm,	Y =   282.441  mm,	Z =   502.065  mm,
	W =   -15.171 deg,	P =   -43.175 deg,	R =    33.524 deg
   GP2:
	UF : 1, UT : 1,
	J1=    90.000 deg,	J2=     0.000 deg
};
P[94]{
   GP1:
	UF : 1, UT : 1,		CONFIG : 'N U B, 0, 0, 0',
	X =   356.016  mm,	Y =    -2.054  mm,	Z =  2424.089  mm,
	W =      .020 deg,	P =   -40.008 deg,	R =     -.011 deg
   GP2:
	UF : 1, UT : 1,
	J1=    80.000 deg,	J2=   -90.000 deg
};
P[95]{
   GP1:
	UF : 1, UT : 1,		CONFIG : 'N U T, 0, 0, 1',
	X =  1917.622  mm,	Y =   283.121  mm,	Z =   189.834  mm,
	W =   -26.631 deg,	P =    72.567 deg,	R =   160.596 deg
   GP2:
	UF : 1, UT : 1,
	J1=    80.000 deg,	J2=   -90.000 deg
};
P[96]{
   GP1:
	UF : 1, UT : 1,		CONFIG : 'N U T, 0, 0, 0',
	X =  2368.673  mm,	Y =    45.599  mm,	Z =  1002.320  mm,
	W =     -.010 deg,	P =    44.998 deg,	R =    66.715 deg
   GP2:
	UF : 1, UT : 1,
	J1=    90.000 deg,	J2=    90.000 deg
};
P[97]{
   GP1:
	UF : 1, UT : 1,		CONFIG : 'N U T, 0, 0, 0',
	X =  1913.400  mm,	Y = -1217.274  mm,	Z =  1258.765  mm,
	W =   -40.515 deg,	P =     2.084 deg,	R =   -24.296 deg
   GP2:
	UF : 1, UT : 1,
	J1=   180.000 deg,	J2=   -90.000 deg
};
P[98]{
   GP1:
	UF : 1, UT : 1,		CONFIG : 'N U T, 0, 0, 0',
	X =  2339.221  mm,	Y =   -53.197  mm,	Z =   838.927  mm,
	W =     4.731 deg,	P =    44.801 deg,	R =    66.707 deg
   GP2:
	UF : 1, UT : 1,
	J1=    90.000 deg,	J2=    90.000 deg
};
P[99]{
   GP1:
	UF : 1, UT : 1,		CONFIG : 'N U T, 0, 0, 0',
	X =  1419.375  mm,	Y =   870.775  mm,	Z =  1903.281  mm,
	W =    32.261 deg,	P =   -18.474 deg,	R =    10.214 deg
   GP2:
	UF : 1, UT : 1,
	J1=   180.000 deg,	J2=    90.000 deg
};
P[100]{
   GP1:
	UF : 1, UT : 1,		CONFIG : 'F U T, 0, 0, 0',
	X =  2701.500  mm,	Y =   248.797  mm,	Z =   650.852  mm,
	W =    -2.629 deg,	P =   -43.936 deg,	R =    42.269 deg
   GP2:
	UF : 1, UT : 1,
	J1=    90.000 deg,	J2=     0.000 deg
};
P[101]{
   GP1:
	UF : 1, UT : 1,		CONFIG : 'N U T, 0, 0, 0',
	X =  2410.572  mm,	Y =   -92.153  mm,	Z =   838.891  mm,
	W =     4.736 deg,	P =    44.800 deg,	R =    66.708 deg
   GP2:
	UF : 1, UT : 1,
	J1=    90.000 deg,	J2=    90.000 deg
};
P[102]{
   GP1:
	UF : 1, UT : 1,		CONFIG : 'N U T, 0, 0, 0',
	X =  2687.056  mm,	Y =  -231.345  mm,	Z =   639.889  mm,
	W =    14.883 deg,	P =   -42.517 deg,	R =   -27.206 deg
   GP2:
	UF : 1, UT : 1,
	J1=    90.000 deg,	J2=     0.000 deg
};
P[103]{
   GP1:
	UF : 1, UT : 1,		CONFIG : 'N U T, 0, 0, 0',
	X =  2860.056  mm,	Y =  -309.345  mm,	Z =   520.586  mm,
	W =    14.883 deg,	P =   -42.517 deg,	R =   -27.206 deg
   GP2:
	UF : 1, UT : 1,
	J1=    90.000 deg,	J2=     0.000 deg
};
P[104]{
   GP1:
	UF : 1, UT : 1,		CONFIG : 'N U B, 0, 0, 0',
	X =   356.007  mm,	Y =    -2.068  mm,	Z =  2424.055  mm,
	W =      .010 deg,	P =   -40.003 deg,	R =     -.004 deg
   GP2:
	UF : 1, UT : 1,
	J1=   180.000 deg,	J2=   150.000 deg
};
P[105]{
   GP1:
	UF : 1, UT : 1,		CONFIG : 'N U T, 0, 0, 0',
	X =  1166.553  mm,	Y = -1374.013  mm,	Z =  1522.225  mm,
	W =   -32.586 deg,	P =   -12.067 deg,	R =    17.529 deg
   GP2:
	UF : 1, UT : 1,
	J1=   180.000 deg,	J2=  -125.000 deg
};
P[106]{
   GP1:
	UF : 1, UT : 1,
	J1=   -55.000 deg,	J2=   -30.678 deg,	J3=    10.000 deg,
	J4=   -84.542 deg,	J5=   -72.333 deg,	J6=   125.863 deg
   GP2:
	UF : 1, UT : 1,
	J1=   100.000 deg,	J2=   -90.000 deg
};
P[107]{
   GP1:
	UF : 1, UT : 1,		CONFIG : 'N U T, 0, 0, 0',
	X =  2337.765  mm,	Y = -1447.908  mm,	Z =  1189.179  mm,
	W =   -45.668 deg,	P =   -29.178 deg,	R =    61.340 deg
   GP2:
	UF : 1, UT : 1,
	J1=   100.000 deg,	J2=   -90.000 deg
};
P[108]{
   GP1:
	UF : 1, UT : 1,		CONFIG : 'N U T, 0, 0, -1',
	X =  2500.465  mm,	Y = -1499.903  mm,	Z =  1059.350  mm,
	W =   -50.284 deg,	P =   -30.325 deg,	R =    67.097 deg
   GP2:
	UF : 0, UT : 1,
	J1=   100.000 deg,	J2=   -90.000 deg
};
P[109]{
   GP1:
	UF : 1, UT : 1,		CONFIG : 'N U T, 0, 0, 0',
	X =  2791.272  mm,	Y = -1482.457  mm,	Z =   932.389  mm,
	W =   -37.771 deg,	P =   -31.405 deg,	R =    42.828 deg
   GP2:
	UF : 1, UT : 1,
	J1=   100.000 deg,	J2=   -90.000 deg
};
P[110]{
   GP1:
	UF : 1, UT : 1,		CONFIG : 'N U T, 0, 0, 0',
	X =  2690.549  mm,	Y =  -310.856  mm,	Z =   600.282  mm,
	W =     1.613 deg,	P =   -43.868 deg,	R =   -40.404 deg
   GP2:
	UF : 1, UT : 1,
	J1=    90.000 deg,	J2=     0.000 deg
};
P[111]{
   GP1:
	UF : 1, UT : 1,		CONFIG : 'N U T, 1, 0, 0',
	X =  2528.555  mm,	Y =   -65.615  mm,	Z =   892.718  mm,
	W =   -11.578 deg,	P =   -57.733 deg,	R =     8.895 deg
   GP2:
	UF : 1, UT : 1,
	J1=    90.000 deg,	J2=     0.000 deg
};
P[112]{
   GP1:
	UF : 1, UT : 1,		CONFIG : 'N U T, 0, 0, 0',
	X =  2860.056  mm,	Y =  -309.345  mm,	Z =   520.586  mm,
	W =    14.883 deg,	P =   -42.517 deg,	R =   -27.206 deg
   GP2:
	UF : 1, UT : 1,
	J1=    90.000 deg,	J2=     0.000 deg
};
P[113]{
   GP1:
	UF : 1, UT : 1,		CONFIG : 'N U T, 0, 0, 0',
	X =  1539.625  mm,	Y = -1470.562  mm,	Z =  1075.975  mm,
	W =   -42.854 deg,	P =   -15.295 deg,	R =    39.123 deg
   GP2:
	UF : 1, UT : 1,
	J1=   180.000 deg,	J2=  -125.000 deg
};
P[114]{
   GP1:
	UF : 1, UT : 1,		CONFIG : 'N U T, 0, 0, 0',
	X =  1851.900  mm,	Y =  1480.079  mm,	Z =  1370.284  mm,
	W =   -15.089 deg,	P =   -28.874 deg,	R =    15.571 deg
   GP2:
	UF : 1, UT : 1,
	J1=    93.119 deg,	J2=    90.000 deg
};
P[115]{
   GP1:
	UF : 1, UT : 1,		CONFIG : 'N U T, 0, 0, 0',
	X =  2526.820  mm,	Y =  1556.392  mm,	Z =  1079.609  mm,
	W =    21.780 deg,	P =   -40.404 deg,	R =   -29.962 deg
   GP2:
	UF : 0, UT : 1,
	J1=    95.000 deg,	J2=    90.000 deg
};
P[116]{
   GP1:
	UF : 1, UT : 1,		CONFIG : 'N U B, 0, 0, 0',
	X =   356.004  mm,	Y =    -2.058  mm,	Z =  2424.066  mm,
	W =      .021 deg,	P =   -40.005 deg,	R =     -.012 deg
   GP2:
	UF : 1, UT : 1,
	J1=   125.000 deg,	J2=     0.000 deg
};
P[117]{
   GP1:
	UF : 1, UT : 1,		CONFIG : 'N U B, 0, 0, 0',
	X =   356.032  mm,	Y =    -2.146  mm,	Z =  2424.050  mm,
	W =      .001 deg,	P =   -40.002 deg,	R =     -.005 deg
   GP2:
	UF : 1, UT : 1,
	J1=     0.000 deg,	J2=   180.000 deg
};
P[118]{
   GP1:
	UF : 1, UT : 1,		CONFIG : 'N U T, 0, 0, 0',
	X =  1214.806  mm,	Y =   169.341  mm,	Z =   386.823  mm,
	W =    23.939 deg,	P =    39.314 deg,	R =  -177.488 deg
   GP2:
	UF : 1, UT : 1,
	J1=    80.000 deg,	J2=   -90.000 deg
};
P[119]{
   GP1:
	UF : 1, UT : 1,		CONFIG : 'N U T, 0, 0, 0',
	X =  2690.549  mm,	Y =  -310.856  mm,	Z =   600.282  mm,
	W =     1.613 deg,	P =   -43.868 deg,	R =   -40.404 deg
   GP2:
	UF : 1, UT : 1,
	J1=    90.000 deg,	J2=     0.000 deg
};
P[120]{
   GP1:
	UF : 1, UT : 1,		CONFIG : 'N U T, 0, 0, 0',
	X =  2420.268  mm,	Y =   -62.420  mm,	Z =   888.262  mm,
	W =     4.742 deg,	P =    44.802 deg,	R =    66.709 deg
   GP2:
	UF : 1, UT : 1,
	J1=    89.999 deg,	J2=    90.000 deg
};
P[121]{
   GP1:
	UF : 1, UT : 1,		CONFIG : 'N U T, 0, 0, -1',
	X =  2671.361  mm,	Y =  -220.509  mm,	Z =   618.788  mm,
	W =    39.952 deg,	P =    49.905 deg,	R =  -159.452 deg
   GP2:
	UF : 1, UT : 1,
	J1=    90.000 deg,	J2=     0.000 deg
};
P[122]{
   GP1:
	UF : 1, UT : 1,		CONFIG : 'N U T, 0, 0, 0',
	X =  2675.436  mm,	Y =  -298.605  mm,	Z =   591.354  mm,
	W =    31.909 deg,	P =    33.590 deg,	R =  -130.034 deg
   GP2:
	UF : 1, UT : 1,
	J1=    90.000 deg,	J2=     0.000 deg
};
P[123]{
   GP1:
	UF : 1, UT : 1,		CONFIG : 'N U T, 0, 0, 0',
	X =  2434.487  mm,	Y =  -113.503  mm,	Z =   886.043  mm,
	W =   -16.311 deg,	P =    44.679 deg,	R =   -47.493 deg
   GP2:
	UF : 1, UT : 1,
	J1=    90.000 deg,	J2=    90.000 deg
};
P[124]{
   GP1:
	UF : 1, UT : 1,		CONFIG : 'N U T, 0, 0, 0',
	X =  2409.251  mm,	Y =   -94.162  mm,	Z =   839.133  mm,
	W =   -16.311 deg,	P =    44.679 deg,	R =   -47.493 deg
   GP2:
	UF : 1, UT : 1,
	J1=    90.000 deg,	J2=    90.000 deg
};
P[125]{
   GP1:
	UF : 1, UT : 1,		CONFIG : 'N U T, 0, 0, 0',
	X =  2394.251  mm,	Y =  -118.758  mm,	Z =   838.191  mm,
	W =   -16.304 deg,	P =    44.678 deg,	R =   -47.499 deg
   GP2:
	UF : 1, UT : 1,
	J1=    90.000 deg,	J2=    90.000 deg
};
P[126]{
   GP1:
	UF : 1, UT : 1,		CONFIG : 'N U T, 0, 0, 0',
	X =  2420.624  mm,	Y =  -138.635  mm,	Z =   886.232  mm,
	W =   -16.306 deg,	P =    44.680 deg,	R =   -47.506 deg
   GP2:
	UF : 1, UT : 1,
	J1=    90.000 deg,	J2=    90.000 deg
};
P[127]{
   GP1:
	UF : 1, UT : 1,		CONFIG : 'N U T, 0, 0, 1',
	X =  2781.845  mm,	Y =  -368.449  mm,	Z =   566.925  mm,
	W =    32.749 deg,	P =    20.905 deg,	R =  -102.080 deg
   GP2:
	UF : 1, UT : 1,
	J1=    90.000 deg,	J2=     0.000 deg
};
P[128]{
   GP1:
	UF : 1, UT : 1,		CONFIG : 'N U T, 0, 0, 0',
	X =  2698.335  mm,	Y =   256.194  mm,	Z =   573.763  mm,
	W =   -42.051 deg,	P =    32.739 deg,	R =   124.663 deg
   GP2:
	UF : 1, UT : 1,
	J1=    90.000 deg,	J2=     0.000 deg
};
P[129]{
   GP1:
	UF : 1, UT : 1,		CONFIG : 'N U T, 0, 0, 0',
	X =  2284.980  mm,	Y =  -119.488  mm,	Z =   927.926  mm,
	W =    34.022 deg,	P =    31.444 deg,	R =   -66.610 deg
   GP2:
	UF : 1, UT : 1,
	J1=    90.000 deg,	J2=    90.000 deg
};
P[130]{
   GP1:
	UF : 1, UT : 1,		CONFIG : 'N U T, 0, 0, 0',
	X =  2325.665  mm,	Y =   -81.955  mm,	Z =   837.767  mm,
	W =    34.413 deg,	P =    31.013 deg,	R =   -66.957 deg
   GP2:
	UF : 1, UT : 1,
	J1=    90.000 deg,	J2=    90.000 deg
};
P[131]{
   GP1:
	UF : 1, UT : 1,		CONFIG : 'N U T, 0, 0, 0',
	X =  2385.550  mm,	Y =  -116.407  mm,	Z =   839.070  mm,
	W =    34.407 deg,	P =    31.012 deg,	R =   -66.953 deg
   GP2:
	UF : 1, UT : 1,
	J1=    90.000 deg,	J2=    90.000 deg
};
P[132]{
   GP1:
	UF : 1, UT : 1,		CONFIG : 'N U T, 0, 0, 0',
	X =  2364.441  mm,	Y =  -140.196  mm,	Z =   874.079  mm,
	W =    33.535 deg,	P =    29.220 deg,	R =   -67.391 deg
   GP2:
	UF : 1, UT : 1,
	J1=    90.000 deg,	J2=    90.000 deg
};
P[133]{
   GP1:
	UF : 1, UT : 1,		CONFIG : 'N U T, 0, 0, 0',
	X =  2750.496  mm,	Y =   369.295  mm,	Z =   531.685  mm,
	W =   -32.204 deg,	P =    27.169 deg,	R =   115.020 deg
   GP2:
	UF : 1, UT : 1,
	J1=    90.000 deg,	J2=     0.000 deg
};
P[134]{
   GP1:
	UF : 1, UT : 1,		CONFIG : 'N U T, 0, 0, 0',
	X =  2433.364  mm,	Y =   -19.547  mm,	Z =   530.114  mm,
	W =    -7.526 deg,	P =    51.572 deg,	R =   125.549 deg
   GP2:
	UF : 1, UT : 1,
	J1=    90.000 deg,	J2=     0.000 deg
};
P[135]{
   GP1:
	UF : 1, UT : 1,		CONFIG : 'N U T, 0, 0, 0',
	X =  1964.092  mm,	Y =   128.072  mm,	Z =   485.282  mm,
	W =    14.025 deg,	P =    31.485 deg,	R =    29.572 deg
   GP2:
	UF : 1, UT : 1,
	J1=    90.000 deg,	J2=     0.000 deg
};
P[136]{
   GP1:
	UF : 1, UT : 1,		CONFIG : 'N U T, 0, 0, 0',
	X =  1776.950  mm,	Y =   181.788  mm,	Z =   449.993  mm,
	W =    35.022 deg,	P =    36.482 deg,	R =    50.220 deg
   GP2:
	UF : 1, UT : 1,
	J1=    90.000 deg,	J2=     0.000 deg
};
P[137]{
   GP1:
	UF : 1, UT : 1,		CONFIG : 'N U T, 0, 0, 0',
	X =  1110.996  mm,	Y =   547.835  mm,	Z =  1204.956  mm,
	W =    30.412 deg,	P =    23.153 deg,	R =   -68.803 deg
   GP2:
	UF : 1, UT : 1,
	J1=    90.000 deg,	J2=    90.000 deg
};
P[138]{
   GP1:
	UF : 1, UT : 1,		CONFIG : 'N U T, 0, 0, 0',
	X =  1746.082  mm,	Y =   249.573  mm,	Z =   569.263  mm,
	W =   -35.537 deg,	P =   -12.977 deg,	R =   -27.038 deg
   GP2:
	UF : 1, UT : 1,
	J1=    90.000 deg,	J2=   100.000 deg
};
P[139]{
   GP1:
	UF : 1, UT : 1,		CONFIG : 'N U T, 0, 0, 0',
	X =  1754.079  mm,	Y =   165.415  mm,	Z =   449.266  mm,
	W =    31.721 deg,	P =    33.769 deg,	R =    48.036 deg
   GP2:
	UF : 1, UT : 1,
	J1=    90.000 deg,	J2=     0.000 deg
};
P[140]{
   GP1:
	UF : 1, UT : 1,		CONFIG : 'N U T, 0, 0, 0',
	X =  1754.079  mm,	Y =  -235.814  mm,	Z =   449.266  mm,
	W =   -34.074 deg,	P =    31.387 deg,	R =   -52.404 deg
   GP2:
	UF : 1, UT : 1,
	J1=    90.000 deg,	J2=     0.000 deg
};
P[141]{
   GP1:
	UF : 1, UT : 1,		CONFIG : 'N U T, 0, 0, 0',
	X =  2157.996  mm,	Y =    56.121  mm,	Z =   156.955  mm,
	W =   -33.684 deg,	P =   -17.646 deg,	R =   -34.041 deg
   GP2:
	UF : 1, UT : 1,
	J1=    90.000 deg,	J2=   100.000 deg
};
P[142]{
   GP1:
	UF : 1, UT : 1,		CONFIG : 'N U T, 0, 0, 0',
	X =  2482.996  mm,	Y =    56.121  mm,	Z =   156.955  mm,
	W =   -33.684 deg,	P =   -17.646 deg,	R =   -34.041 deg
   GP2:
	UF : 1, UT : 1,
	J1=    90.000 deg,	J2=   100.000 deg
};
P[143]{
   GP1:
	UF : 1, UT : 1,		CONFIG : 'N U T, 0, 0, 0',
	X =  1843.198  mm,	Y =  -173.825  mm,	Z =   537.934  mm,
	W =   -34.074 deg,	P =    31.387 deg,	R =   -52.404 deg
   GP2:
	UF : 1, UT : 1,
	J1=    90.000 deg,	J2=     0.000 deg
};
P[144]{
   GP1:
	UF : 1, UT : 1,		CONFIG : 'N U T, 0, 0, 0',
	X =  1807.054  mm,	Y =   -90.826  mm,	Z =  1125.220  mm,
	W =      .036 deg,	P =     1.106 deg,	R =     1.891 deg
   GP2:
	UF : 1, UT : 1,
	J1=    45.000 deg,	J2=     0.000 deg
};
P[145]{
   GP1:
	UF : 1, UT : 1,		CONFIG : 'N U T, 0, 0, 0',
	X =  1807.054  mm,	Y =  -390.825  mm,	Z =  1004.220  mm,
	W =     -.607 deg,	P =      .924 deg,	R =   -33.344 deg
   GP2:
	UF : 1, UT : 1,
	J1=    45.000 deg,	J2=     0.000 deg
};
P[146]{
   GP1:
	UF : 1, UT : 1,		CONFIG : 'N U T, 0, 0, 0',
	X =  2520.811  mm,	Y =   -87.819  mm,	Z =   -31.343  mm,
	W =   -31.347 deg,	P =   -16.435 deg,	R =   -28.772 deg
   GP2:
	UF : 1, UT : 1,
	J1=    90.000 deg,	J2=   100.000 deg
};
P[147]{
   GP1:
	UF : 1, UT : 1,		CONFIG : 'N U T, 0, 0, 0',
	X =  2476.165  mm,	Y =   -87.819  mm,	Z =   -31.343  mm,
	W =   -31.347 deg,	P =   -16.435 deg,	R =   -32.491 deg
   GP2:
	UF : 1, UT : 1,
	J1=    90.000 deg,	J2=   100.000 deg
};
P[148]{
   GP1:
	UF : 1, UT : 1,		CONFIG : 'N U T, 0, 0, 0',
	X =  1816.054  mm,	Y =  -176.826  mm,	Z =  1084.220  mm,
	W =     -.607 deg,	P =      .924 deg,	R =   -33.344 deg
   GP2:
	UF : 1, UT : 1,
	J1=    45.000 deg,	J2=     0.000 deg
};
P[149]{
   GP1:
	UF : 1, UT : 1,		CONFIG : 'N U T, 0, 0, 0',
	X =  1807.054  mm,	Y =   376.174  mm,	Z =  1018.220  mm,
	W =     -.607 deg,	P =      .924 deg,	R =    40.441 deg
   GP2:
	UF : 1, UT : 1,
	J1=    45.000 deg,	J2=     0.000 deg
};
P[150]{
   GP1:
	UF : 1, UT : 1,		CONFIG : 'N U T, 0, 0, 0',
	X =  2445.324  mm,	Y =   -88.013  mm,	Z =   -29.938  mm,
	W =   -31.347 deg,	P =   -16.435 deg,	R =   -51.724 deg
   GP2:
	UF : 1, UT : 1,
	J1=    90.000 deg,	J2=   100.000 deg
};
P[151]{
   GP1:
	UF : 1, UT : 1,		CONFIG : 'N U T, 0, 0, 0',
	X =  2550.156  mm,	Y =    45.835  mm,	Z =   135.483  mm,
	W =   -31.566 deg,	P =   -16.651 deg,	R =   -48.456 deg
   GP2:
	UF : 1, UT : 1,
	J1=    90.000 deg,	J2=   100.000 deg
};
P[152]{
   GP1:
	UF : 1, UT : 1,		CONFIG : 'N U T, 0, 0, 0',
	X =  1807.054  mm,	Y =   173.895  mm,	Z =  1166.219  mm,
	W =     -.607 deg,	P =      .924 deg,	R =    40.441 deg
   GP2:
	UF : 1, UT : 1,
	J1=    45.000 deg,	J2=     0.000 deg
};
P[153]{
   GP1:
	UF : 1, UT : 1,		CONFIG : 'N U T, 0, 0, 0',
	X =   908.243  mm,	Y =     -.972  mm,	Z =  2177.323  mm,
	W =     -.010 deg,	P =   -45.000 deg,	R =     0.000 deg
   GP2:
	UF : 1, UT : 1,
	J1=   125.000 deg,	J2=     0.000 deg
};
P[154]{
   GP1:
	UF : 1, UT : 1,		CONFIG : 'N U T, 0, 0, 0',
	X =  1841.244  mm,	Y =   574.028  mm,	Z =  1589.322  mm,
	W =     -.010 deg,	P =   -11.091 deg,	R =     0.000 deg
   GP2:
	UF : 1, UT : 1,
	J1=   125.000 deg,	J2=     0.000 deg
};
P[155]{
   GP1:
	UF : 1, UT : 1,		CONFIG : 'N U T, 0, 0, 0',
	X =  2130.244  mm,	Y =   574.028  mm,	Z =  1472.322  mm,
	W =     -.010 deg,	P =   -11.091 deg,	R =     0.000 deg
   GP2:
	UF : 1, UT : 1,
	J1=   125.000 deg,	J2=     0.000 deg
};
P[156]{
   GP1:
	UF : 1, UT : 1,		CONFIG : 'N U T, 0, 0, 0',
	X =  2346.710  mm,	Y =    66.661  mm,	Z =   156.955  mm,
	W =   -33.684 deg,	P =   -17.646 deg,	R =   -34.041 deg
   GP2:
	UF : 1, UT : 1,
	J1=    90.000 deg,	J2=   100.000 deg
};
P[157]{
   GP1:
	UF : 1, UT : 1,		CONFIG : 'N U T, 0, 0, 0',
	X =  2346.283  mm,	Y =   -84.749  mm,	Z =   -32.121  mm,
	W =   -31.932 deg,	P =   -15.149 deg,	R =   -19.992 deg
   GP2:
	UF : 1, UT : 1,
	J1=    90.000 deg,	J2=   100.000 deg
};
P[158]{
   GP1:
	UF : 1, UT : 1,		CONFIG : 'N U T, 0, 0, 0',
	X =  2395.638  mm,	Y =   -85.392  mm,	Z =   -32.121  mm,
	W =   -31.932 deg,	P =   -15.149 deg,	R =   -19.992 deg
   GP2:
	UF : 1, UT : 1,
	J1=    90.000 deg,	J2=   100.000 deg
};
P[159]{
   GP1:
	UF : 1, UT : 1,		CONFIG : 'N U T, 0, 0, 0',
	X =  2192.055  mm,	Y =   448.511  mm,	Z =  1378.272  mm,
	W =     0.000 deg,	P =    -1.567 deg,	R =     0.000 deg
   GP2:
	UF : 1, UT : 1,
	J1=   125.000 deg,	J2=     0.000 deg
};
P[160]{
   GP1:
	UF : 1, UT : 1,		CONFIG : 'N U T, 0, 0, 0',
	X =  2174.054  mm,	Y =    17.763  mm,	Z =  1379.272  mm,
	W =     0.000 deg,	P =    -1.567 deg,	R =     0.000 deg
   GP2:
	UF : 1, UT : 1,
	J1=   125.000 deg,	J2=     0.000 deg
};
P[161]{
   GP1:
	UF : 1, UT : 1,		CONFIG : 'N U T, 0, 0, 1',
	X =  2740.275  mm,	Y =  -288.449  mm,	Z =   453.193  mm,
	W =    32.535 deg,	P =    32.993 deg,	R =  -130.484 deg
   GP2:
	UF : 1, UT : 1,
	J1=    90.000 deg,	J2=     0.000 deg
};
P[162]{
   GP1:
	UF : 1, UT : 1,		CONFIG : 'N U T, 0, 0, 1',
	X =  2739.668  mm,	Y =  -336.172  mm,	Z =   453.798  mm,
	W =    32.535 deg,	P =    32.993 deg,	R =  -130.484 deg
   GP2:
	UF : 1, UT : 1,
	J1=    90.000 deg,	J2=     0.000 deg
};
P[163]{
   GP1:
	UF : 1, UT : 1,		CONFIG : 'N U T, 0, 0, 0',
	X =  2194.122  mm,	Y =  -401.237  mm,	Z =  1396.402  mm,
	W =     0.000 deg,	P =     1.835 deg,	R =     0.000 deg
   GP2:
	UF : 1, UT : 1,
	J1=   125.000 deg,	J2=     0.000 deg
};
P[164]{
   GP1:
	UF : 1, UT : 1,		CONFIG : 'N U T, 0, 0, 0',
	X =  2176.122  mm,	Y =   354.763  mm,	Z =  1397.402  mm,
	W =     0.000 deg,	P =     1.835 deg,	R =     0.000 deg
   GP2:
	UF : 1, UT : 1,
	J1=   125.000 deg,	J2=     0.000 deg
};
P[165]{
   GP1:
	UF : 1, UT : 1,		CONFIG : 'N U T, 0, 0, 1',
	X =  2758.004  mm,	Y =  -362.559  mm,	Z =   454.194  mm,
	W =    32.708 deg,	P =    26.756 deg,	R =  -103.211 deg
   GP2:
	UF : 1, UT : 1,
	J1=    90.000 deg,	J2=     0.000 deg
};
P[166]{
   GP1:
	UF : 1, UT : 1,		CONFIG : 'N U T, 0, 0, 1',
	X =  2775.874  mm,	Y =  -366.475  mm,	Z =   454.510  mm,
	W =    32.938 deg,	P =    19.373 deg,	R =   -84.969 deg
   GP2:
	UF : 1, UT : 1,
	J1=    90.000 deg,	J2=     0.000 deg
};
P[167]{
   GP1:
	UF : 1, UT : 1,		CONFIG : 'N U T, 0, 0, 0',
	X =  2176.122  mm,	Y =    15.763  mm,	Z =  1427.402  mm,
	W =     0.000 deg,	P =    -4.591 deg,	R =     0.000 deg
   GP2:
	UF : 1, UT : 1,
	J1=   125.000 deg,	J2=     0.000 deg
};
P[168]{
   GP1:
	UF : 1, UT : 1,		CONFIG : 'N U T, 0, 0, 0',
	X =  2176.122  mm,	Y =  -553.165  mm,	Z =  1427.402  mm,
	W =     0.000 deg,	P =    -4.591 deg,	R =     0.000 deg
   GP2:
	UF : 1, UT : 1,
	J1=   125.000 deg,	J2=     0.000 deg
};
P[169]{
   GP1:
	UF : 1, UT : 1,		CONFIG : 'N U T, 0, 0, 0',
	X =  2738.871  mm,	Y =   286.873  mm,	Z =   453.249  mm,
	W =   -36.613 deg,	P =    28.244 deg,	R =   122.493 deg
   GP2:
	UF : 1, UT : 1,
	J1=    90.000 deg,	J2=     0.000 deg
};
P[170]{
   GP1:
	UF : 1, UT : 1,		CONFIG : 'N U T, 0, 0, 0',
	X =  2739.301  mm,	Y =   336.925  mm,	Z =   453.098  mm,
	W =   -36.613 deg,	P =    28.244 deg,	R =   122.493 deg
   GP2:
	UF : 1, UT : 1,
	J1=    90.000 deg,	J2=     0.000 deg
};
P[171]{
   GP1:
	UF : 1, UT : 1,		CONFIG : 'N U T, 0, 0, 0',
	X =  2758.115  mm,	Y =   360.338  mm,	Z =   452.692  mm,
	W =   -32.204 deg,	P =    27.169 deg,	R =   100.051 deg
   GP2:
	UF : 1, UT : 1,
	J1=    90.000 deg,	J2=     0.000 deg
};
P[172]{
   GP1:
	UF : 1, UT : 1,		CONFIG : 'N U T, 0, 0, 0',
	X =  2174.639  mm,	Y =  -639.399  mm,	Z =  1514.172  mm,
	W =     0.000 deg,	P =   -23.113 deg,	R =     0.000 deg
   GP2:
	UF : 1, UT : 1,
	J1=   125.000 deg,	J2=     0.000 deg
};
P[173]{
   GP1:
	UF : 1, UT : 1,		CONFIG : 'N U T, 0, 0, 0',
	X =  1929.795  mm,	Y =  -639.399  mm,	Z =  1514.172  mm,
	W =     0.000 deg,	P =   -23.113 deg,	R =     0.000 deg
   GP2:
	UF : 1, UT : 1,
	J1=   125.000 deg,	J2=     0.000 deg
};
P[174]{
   GP1:
	UF : 1, UT : 1,		CONFIG : 'N U B, 0, 0, 0',
	X =   356.032  mm,	Y =    -2.146  mm,	Z =  2424.050  mm,
	W =      .001 deg,	P =   -40.002 deg,	R =     -.005 deg
   GP2:
	UF : 1, UT : 1,
	J1=     0.000 deg,	J2=   180.000 deg
};
P[175]{
   GP1:
	UF : 1, UT : 1,		CONFIG : 'N U T, 0, 0, 0',
	X =   908.243  mm,	Y =     -.972  mm,	Z =  1061.322  mm,
	W =     -.010 deg,	P =    45.000 deg,	R =   -90.656 deg
   GP2:
	UF : 1, UT : 1,
	J1=     0.000 deg,	J2=   180.000 deg
};
P[176]{
   GP1:
	UF : 1, UT : 1,		CONFIG : 'N U T, 0, 0, 0',
	X =  2167.744  mm,	Y =   245.457  mm,	Z =   371.894  mm,
	W =    34.980 deg,	P =    30.342 deg,	R =   -11.521 deg
   GP2:
	UF : 1, UT : 1,
	J1=     0.000 deg,	J2=   180.000 deg
};
P[177]{
   GP1:
	UF : 1, UT : 1,		CONFIG : 'N U T, 0, 0, 0',
	X =  2773.933  mm,	Y =   364.055  mm,	Z =   454.486  mm,
	W =   -28.529 deg,	P =    23.417 deg,	R =    94.769 deg
   GP2:
	UF : 1, UT : 1,
	J1=    90.000 deg,	J2=     0.000 deg
};
P[178]{
   GP1:
	UF : 1, UT : 1,		CONFIG : 'N U T, 0, 0, 0',
	X =  1666.536  mm,	Y =   240.508  mm,	Z =   356.880  mm,
	W =    31.721 deg,	P =    33.769 deg,	R =    50.168 deg
   GP2:
	UF : 1, UT : 1,
	J1=    90.000 deg,	J2=     0.000 deg
};
P[179]{
   GP1:
	UF : 1, UT : 1,		CONFIG : 'N U T, 0, 0, 0',
	X =  1665.250  mm,	Y =   163.365  mm,	Z =   356.880  mm,
	W =    31.721 deg,	P =    33.769 deg,	R =    50.168 deg
   GP2:
	UF : 1, UT : 1,
	J1=    90.000 deg,	J2=     0.000 deg
};
P[180]{
   GP1:
	UF : 1, UT : 1,		CONFIG : 'N U T, 0, 0, 0',
	X =  1670.256  mm,	Y =  -244.713  mm,	Z =   361.510  mm,
	W =   -34.074 deg,	P =    31.387 deg,	R =   -56.109 deg
   GP2:
	UF : 1, UT : 1,
	J1=    90.000 deg,	J2=     0.000 deg
};
P[181]{
   GP1:
	UF : 1, UT : 1,		CONFIG : 'N U T, 0, 0, 0',
	X =  2189.474  mm,	Y =   383.790  mm,	Z =   296.220  mm,
	W =    47.745 deg,	P =     8.599 deg,	R =   -35.895 deg
   GP2:
	UF : 1, UT : 1,
	J1=     0.000 deg,	J2=   180.000 deg
};
P[182]{
   GP1:
	UF : 1, UT : 1,		CONFIG : 'N U T, 0, 0, 0',
	X =  2150.796  mm,	Y =    51.228  mm,	Z =   379.826  mm,
	W =     9.396 deg,	P =    -3.028 deg,	R =   -24.284 deg
   GP2:
	UF : 1, UT : 1,
	J1=     0.000 deg,	J2=   180.000 deg
};
P[183]{
   GP1:
	UF : 1, UT : 1,		CONFIG : 'N U T, 0, 0, 0',
	X =  1058.698  mm,	Y =   195.065  mm,	Z =  1283.367  mm,
	W =    73.635 deg,	P =    26.735 deg,	R =   -73.196 deg
   GP2:
	UF : 1, UT : 1,
	J1=   -90.000 deg,	J2=   -90.000 deg
};
P[184]{
   GP1:
	UF : 1, UT : 1,		CONFIG : 'N U T, 0, 0, 0',
	X =  2161.838  mm,	Y =  -354.344  mm,	Z =   373.103  mm,
	W =   -42.503 deg,	P =    -2.383 deg,	R =   -32.742 deg
   GP2:
	UF : 1, UT : 1,
	J1=     0.000 deg,	J2=   180.000 deg
};
P[185]{
   GP1:
	UF : 1, UT : 1,		CONFIG : 'N U T, 0, 0, 0',
	X =  1669.601  mm,	Y =  -166.758  mm,	Z =   359.996  mm,
	W =   -34.074 deg,	P =    31.387 deg,	R =   -56.109 deg
   GP2:
	UF : 1, UT : 1,
	J1=    90.000 deg,	J2=     0.000 deg
};
P[186]{
   GP1:
	UF : 1, UT : 1,		CONFIG : 'N U T, 0, 0, 0',
	X =  1808.487  mm,	Y =  -398.294  mm,	Z =   825.846  mm,
	W =     -.607 deg,	P =      .924 deg,	R =   -33.344 deg
   GP2:
	UF : 1, UT : 1,
	J1=    45.000 deg,	J2=     0.000 deg
};
P[187]{
   GP1:
	UF : 1, UT : 1,		CONFIG : 'N U T, 0, 0, 0',
	X =  1809.130  mm,	Y =  -167.508  mm,	Z =   821.989  mm,
	W =     -.607 deg,	P =      .924 deg,	R =   -33.344 deg
   GP2:
	UF : 1, UT : 1,
	J1=    45.000 deg,	J2=     0.000 deg
};
P[188]{
   GP1:
	UF : 1, UT : 1,		CONFIG : 'N U T, 0, 0, 0',
	X =  1814.471  mm,	Y =   396.122  mm,	Z =   827.314  mm,
	W =     -.603 deg,	P =      .917 deg,	R =    40.436 deg
   GP2:
	UF : 1, UT : 1,
	J1=    45.000 deg,	J2=     0.000 deg
};
P[189]{
   GP1:
	UF : 1, UT : 1,		CONFIG : 'N U T, 0, 0, 0',
	X =  2149.286  mm,	Y =  -279.133  mm,	Z =   456.472  mm,
	W =   -44.186 deg,	P =    -9.562 deg,	R =     3.909 deg
   GP2:
	UF : 1, UT : 1,
	J1=     0.000 deg,	J2=   180.000 deg
};
P[190]{
   GP1:
	UF : 1, UT : 1,		CONFIG : 'N U T, 0, 0, 1',
	X =  1982.724  mm,	Y =   -25.313  mm,	Z =   235.548  mm,
	W =    21.889 deg,	P =    35.316 deg,	R =  -145.925 deg
   GP2:
	UF : 1, UT : 1,
	J1=     0.000 deg,	J2=   180.000 deg
};
P[191]{
   GP1:
	UF : 1, UT : 1,		CONFIG : 'N U T, 0, 0, 1',
	X =  2182.725  mm,	Y =  -216.312  mm,	Z =    -6.136  mm,
	W =    32.857 deg,	P =    25.665 deg,	R =  -124.570 deg
   GP2:
	UF : 1, UT : 1,
	J1=     0.000 deg,	J2=   180.000 deg
};
P[192]{
   GP1:
	UF : 1, UT : 1,		CONFIG : 'N U T, 0, 0, 0',
	X =  1809.837  mm,	Y =   170.236  mm,	Z =   830.044  mm,
	W =     -.606 deg,	P =      .923 deg,	R =    40.441 deg
   GP2:
	UF : 1, UT : 1,
	J1=    45.000 deg,	J2=     0.000 deg
};
P[193]{
   GP1:
	UF : 1, UT : 1,		CONFIG : 'N U T, 0, 0, 0',
	X =  2187.164  mm,	Y =   650.333  mm,	Z =  1313.407  mm,
	W =     -.227 deg,	P =     5.389 deg,	R =     -.013 deg
   GP2:
	UF : 1, UT : 1,
	J1=   125.000 deg,	J2=     0.000 deg
};
P[194]{
   GP1:
	UF : 1, UT : 1,		CONFIG : 'N U T, 0, 0, 0',
	X =  2187.731  mm,	Y =   465.760  mm,	Z =  1315.759  mm,
	W =     0.000 deg,	P =     3.348 deg,	R =     0.000 deg
   GP2:
	UF : 1, UT : 1,
	J1=   125.000 deg,	J2=     0.000 deg
};
P[195]{
   GP1:
	UF : 1, UT : 1,		CONFIG : 'N U T, 0, 0, 1',
	X =  2185.038  mm,	Y =   -47.631  mm,	Z =   -82.880  mm,
	W =     1.218 deg,	P =    44.987 deg,	R =  -147.433 deg
   GP2:
	UF : 1, UT : 1,
	J1=     0.000 deg,	J2=   180.000 deg
};
P[196]{
   GP1:
	UF : 1, UT : 1,		CONFIG : 'N U T, 0, 0, 0',
	X =  2185.038  mm,	Y =   213.369  mm,	Z =   -82.880  mm,
	W =   -26.253 deg,	P =    37.378 deg,	R =   139.534 deg
   GP2:
	UF : 1, UT : 1,
	J1=     0.000 deg,	J2=   180.000 deg
};
P[197]{
   GP1:
	UF : 1, UT : 1,		CONFIG : 'N U T, 0, 0, 0',
	X =  2187.560  mm,	Y =   449.568  mm,	Z =  1316.429  mm,
	W =    -8.764 deg,	P =     3.263 deg,	R =     -.929 deg
   GP2:
	UF : 1, UT : 1,
	J1=   124.998 deg,	J2=     0.000 deg
};
P[198]{
   GP1:
	UF : 1, UT : 1,		CONFIG : 'N U T, 0, 0, 0',
	X =  2174.031  mm,	Y =    21.965  mm,	Z =  1338.187  mm,
	W =     -.928 deg,	P =     6.431 deg,	R =     -.103 deg
   GP2:
	UF : 1, UT : 1,
	J1=   125.000 deg,	J2=     0.000 deg
};
P[199]{
   GP1:
	UF : 1, UT : 1,		CONFIG : 'N U T, 0, 0, 0',
	X =  2170.659  mm,	Y =  -403.519  mm,	Z =  1333.511  mm,
	W =     -.913 deg,	P =     6.529 deg,	R =     -.103 deg
   GP2:
	UF : 1, UT : 1,
	J1=   125.000 deg,	J2=     0.000 deg
};
P[200]{
   GP1:
	UF : 1, UT : 1,		CONFIG : 'N U T, 0, 0, 0',
	X =  2149.428  mm,	Y =    61.346  mm,	Z =   -40.697  mm,
	W =    14.710 deg,	P =    43.024 deg,	R =   172.922 deg
   GP2:
	UF : 1, UT : 1,
	J1=     0.000 deg,	J2=   180.000 deg
};
P[201]{
   GP1:
	UF : 1, UT : 1,		CONFIG : 'N U T, 0, 0, 0',
	X =  1379.179  mm,	Y =     5.048  mm,	Z =   295.119  mm,
	W =    -2.053 deg,	P =    45.296 deg,	R =  -168.776 deg
   GP2:
	UF : 1, UT : 1,
	J1=     0.000 deg,	J2=   180.000 deg
};
P[202]{
   GP1:
	UF : 1, UT : 1,		CONFIG : 'N U T, 0, 0, 1',
	X =  1381.432  mm,	Y =  -574.038  mm,	Z =   156.436  mm,
	W =    42.351 deg,	P =    16.902 deg,	R =  -106.783 deg
   GP2:
	UF : 1, UT : 1,
	J1=     0.000 deg,	J2=   180.000 deg
};
P[203]{
   GP1:
	UF : 1, UT : 1,		CONFIG : 'N U T, 0, 0, 0',
	X =  2174.530  mm,	Y =   403.950  mm,	Z =  1333.813  mm,
	W =    -1.719 deg,	P =     6.202 deg,	R =     -.185 deg
   GP2:
	UF : 1, UT : 1,
	J1=   125.000 deg,	J2=     0.000 deg
};
P[204]{
   GP1:
	UF : 1, UT : 1,		CONFIG : 'N U T, 0, 0, 0',
	X =  2173.957  mm,	Y =    22.391  mm,	Z =  1335.255  mm,
	W =    -1.719 deg,	P =     6.202 deg,	R =     -.185 deg
   GP2:
	UF : 1, UT : 1,
	J1=   125.000 deg,	J2=     0.000 deg
};
P[205]{
   GP1:
	UF : 1, UT : 1,		CONFIG : 'N U T, 0, 0, 0',
	X =  2190.994  mm,	Y =  -644.699  mm,	Z =  1316.261  mm,
	W =     0.000 deg,	P =     5.742 deg,	R =     0.000 deg
   GP2:
	UF : 1, UT : 1,
	J1=   125.000 deg,	J2=     0.000 deg
};
P[206]{
   GP1:
	UF : 1, UT : 1,		CONFIG : 'N U T, 0, 0, 1',
	X =  1351.612  mm,	Y =  -644.118  mm,	Z =   196.361  mm,
	W =    42.489 deg,	P =    16.481 deg,	R =  -107.209 deg
   GP2:
	UF : 1, UT : 1,
	J1=     0.000 deg,	J2=   180.000 deg
};
P[207]{
   GP1:
	UF : 1, UT : 1,		CONFIG : 'N U T, 0, 0, 0',
	X =  1351.612  mm,	Y =     1.774  mm,	Z =   196.362  mm,
	W =     -.786 deg,	P =    44.995 deg,	R =   178.888 deg
   GP2:
	UF : 1, UT : 1,
	J1=     0.000 deg,	J2=   180.000 deg
};
P[208]{
   GP1:
	UF : 1, UT : 1,		CONFIG : 'N U T, 0, 0, 0',
	X =  2184.055  mm,	Y =  -458.842  mm,	Z =  1314.495  mm,
	W =     0.000 deg,	P =     5.742 deg,	R =     0.000 deg
   GP2:
	UF : 1, UT : 1,
	J1=   125.000 deg,	J2=     0.000 deg
};
P[209]{
   GP1:
	UF : 1, UT : 1,		CONFIG : 'N U T, 0, 0, 0',
	X =  2191.159  mm,	Y =  -446.473  mm,	Z =  1319.655  mm,
	W =     4.785 deg,	P =     5.721 deg,	R =      .479 deg
   GP2:
	UF : 1, UT : 1,
	J1=   125.000 deg,	J2=     0.000 deg
};
P[210]{
   GP1:
	UF : 1, UT : 1,		CONFIG : 'N U T, 0, 0, 0',
	X =  1404.034  mm,	Y =  -379.314  mm,	Z =   119.254  mm,
	W =    18.566 deg,	P =    41.762 deg,	R =  -153.239 deg
   GP2:
	UF : 1, UT : 1,
	J1=     0.000 deg,	J2=   180.000 deg
};
P[211]{
   GP1:
	UF : 1, UT : 1,		CONFIG : 'N U T, 0, 0, 0',
	X =  1404.034  mm,	Y =   331.497  mm,	Z =   119.254  mm,
	W =   -20.958 deg,	P =    40.782 deg,	R =   149.612 deg
   GP2:
	UF : 1, UT : 1,
	J1=     0.000 deg,	J2=   180.000 deg
};
P[212]{
   GP1:
	UF : 1, UT : 1,		CONFIG : 'N U T, 0, 0, 0',
	X =  2131.981  mm,	Y =   411.094  mm,	Z =   270.267  mm,
	W =    39.276 deg,	P =    23.852 deg,	R =     9.193 deg
   GP2:
	UF : 1, UT : 1,
	J1=     0.000 deg,	J2=   180.000 deg
};
P[213]{
   GP1:
	UF : 1, UT : 1,		CONFIG : 'N U T, 0, 0, 0',
	X =  2151.123  mm,	Y =   410.023  mm,	Z =   270.268  mm,
	W =    39.276 deg,	P =    23.852 deg,	R =   -24.752 deg
   GP2:
	UF : 1, UT : 1,
	J1=     0.000 deg,	J2=   180.000 deg
};
P[214]{
   GP1:
	UF : 1, UT : 1,		CONFIG : 'N U T, 0, 0, 0',
	X =  1267.764  mm,	Y =    -5.079  mm,	Z =   257.741  mm,
	W =     -.786 deg,	P =    44.995 deg,	R =   178.888 deg
   GP2:
	UF : 1, UT : 1,
	J1=     0.000 deg,	J2=   180.000 deg
};
P[215]{
   GP1:
	UF : 1, UT : 1,		CONFIG : 'N U T, 0, 0, 0',
	X =  1267.763  mm,	Y =   567.064  mm,	Z =   257.741  mm,
	W =    24.666 deg,	P =    38.913 deg,	R =  -143.830 deg
   GP2:
	UF : 1, UT : 1,
	J1=     0.000 deg,	J2=   180.000 deg
};
P[216]{
   GP1:
	UF : 1, UT : 1,		CONFIG : 'N U T, 0, 0, 0',
	X =  2185.123  mm,	Y =   409.594  mm,	Z =   270.268  mm,
	W =    39.276 deg,	P =    23.852 deg,	R =   -24.752 deg
   GP2:
	UF : 1, UT : 1,
	J1=     0.000 deg,	J2=   180.000 deg
};
P[217]{
   GP1:
	UF : 1, UT : 1,		CONFIG : 'N U T, 0, 0, 0',
	X =  2198.754  mm,	Y =   406.887  mm,	Z =   274.717  mm,
	W =    41.358 deg,	P =    19.397 deg,	R =   -47.589 deg
   GP2:
	UF : 1, UT : 1,
	J1=     0.000 deg,	J2=   180.000 deg
};
P[218]{
   GP1:
	UF : 1, UT : 1,		CONFIG : 'N U T, 0, 0, 0',
	X =  2122.108  mm,	Y =  -413.217  mm,	Z =   274.536  mm,
	W =   -42.981 deg,	P =    -2.052 deg,	R =   -39.195 deg
   GP2:
	UF : 1, UT : 1,
	J1=     0.000 deg,	J2=   180.000 deg
};
P[219]{
   GP1:
	UF : 1, UT : 1,		CONFIG : 'N U T, 0, 0, 0',
	X =  1302.181  mm,	Y =   638.659  mm,	Z =   248.465  mm,
	W =    31.136 deg,	P =    34.298 deg,	R =  -133.008 deg
   GP2:
	UF : 1, UT : 1,
	J1=     0.000 deg,	J2=   180.000 deg
};
P[220]{
   GP1:
	UF : 1, UT : 1,		CONFIG : 'N U T, 0, 0, 0',
	X =  1186.272  mm,	Y =   472.511  mm,	Z =   672.833  mm,
	W =    32.440 deg,	P =    45.276 deg,	R =   -70.624 deg
   GP2:
	UF : 1, UT : 1,
	J1=     0.000 deg,	J2=   180.000 deg
};
P[221]{
   GP1:
	UF : 1, UT : 1,		CONFIG : 'N U T, 0, 0, 0',
	X =  2148.036  mm,	Y =  -413.218  mm,	Z =   272.821  mm,
	W =   -42.980 deg,	P =    -2.052 deg,	R =     -.109 deg
   GP2:
	UF : 1, UT : 1,
	J1=     0.000 deg,	J2=   180.000 deg
};
P[222]{
   GP1:
	UF : 1, UT : 1,		CONFIG : 'N U T, 0, 0, 0',
	X =  2187.464  mm,	Y =  -413.218  mm,	Z =   272.821  mm,
	W =   -42.980 deg,	P =    -2.052 deg,	R =     -.109 deg
   GP2:
	UF : 1, UT : 1,
	J1=     0.000 deg,	J2=   180.000 deg
};
P[223]{
   GP1:
	UF : 1, UT : 1,		CONFIG : 'N U T, 0, 0, 0',
	X =  2204.667  mm,	Y =  -410.719  mm,	Z =   275.640  mm,
	W =   -42.298 deg,	P =    -8.712 deg,	R =    19.952 deg
   GP2:
	UF : 1, UT : 1,
	J1=     0.000 deg,	J2=   180.000 deg
};
P[224]{
   GP1:
	UF : 1, UT : 1,		CONFIG : 'N U T, 0, 0, 0',
	X =  1759.654  mm,	Y =  1128.978  mm,	Z =   266.859  mm,
	W =   -16.763 deg,	P =    16.253 deg,	R =    47.184 deg
   GP2:
	UF : 1, UT : 1,
	J1=    90.000 deg,	J2=    90.000 deg
};
P[225]{
   GP1:
	UF : 1, UT : 1,		CONFIG : 'N U T, 0, 0, 0',
	X =  1547.891  mm,	Y =   -77.836  mm,	Z =    80.464  mm,
	W =     5.459 deg,	P =    -9.689 deg,	R =   -27.215 deg
   GP2:
	UF : 1, UT : 1,
	J1=     0.000 deg,	J2=   180.000 deg
};
P[226]{
   GP1:
	UF : 1, UT : 1,		CONFIG : 'N U T, 0, 0, 1',
	X =  2225.517  mm,	Y =  -243.367  mm,	Z =  -199.177  mm,
	W =    34.826 deg,	P =    27.078 deg,	R =  -123.455 deg
   GP2:
	UF : 1, UT : 1,
	J1=     0.000 deg,	J2=   180.000 deg
};
P[227]{
   GP1:
	UF : 1, UT : 1,		CONFIG : 'N U T, 0, 0, 1',
	X =  2225.516  mm,	Y =   -21.581  mm,	Z =  -199.177  mm,
	W =    34.826 deg,	P =    27.077 deg,	R =  -123.454 deg
   GP2:
	UF : 1, UT : 1,
	J1=     0.000 deg,	J2=   180.000 deg
};
P[228]{
   GP1:
	UF : 1, UT : 1,		CONFIG : 'N U T, 0, 0, 1',
	X =  2225.434  mm,	Y =   -11.818  mm,	Z =  -199.807  mm,
	W =    34.761 deg,	P =    27.083 deg,	R =   -99.270 deg
   GP2:
	UF : 1, UT : 1,
	J1=      .000 deg,	J2=   180.000 deg
};
P[229]{
   GP1:
	UF : 1, UT : 1,		CONFIG : 'N U T, 0, 0, 0',
	X =  2223.920  mm,	Y =   250.636  mm,	Z =  -199.420  mm,
	W =   -26.754 deg,	P =    37.334 deg,	R =   139.553 deg
   GP2:
	UF : 1, UT : 1,
	J1=     0.000 deg,	J2=   180.000 deg
};
P[230]{
   GP1:
	UF : 1, UT : 1,		CONFIG : 'N U T, 0, 0, 0',
	X =  1458.812  mm,	Y =  -160.809  mm,	Z =   231.788  mm,
	W =     9.627 deg,	P =   -18.262 deg,	R =   -28.428 deg
   GP2:
	UF : 1, UT : 1,
	J1=     0.000 deg,	J2=   180.000 deg
};
P[231]{
   GP1:
	UF : 1, UT : 1,		CONFIG : 'N U T, 0, 0, 0',
	X =  2848.678  mm,	Y =  1384.540  mm,	Z =   -21.360  mm,
	W =     1.382 deg,	P =      .552 deg,	R =    23.522 deg
   GP2:
	UF : 1, UT : 1,
	J1=    90.000 deg,	J2=    90.000 deg
};
P[232]{
   GP1:
	UF : 1, UT : 1,		CONFIG : 'N U T, 0, 0, 0',
	X =  2848.678  mm,	Y =  1384.540  mm,	Z =   -16.217  mm,
	W =     1.382 deg,	P =      .552 deg,	R =    23.522 deg
   GP2:
	UF : 1, UT : 1,
	J1=    90.000 deg,	J2=    90.000 deg
};
P[233]{
   GP1:
	UF : 1, UT : 1,		CONFIG : 'N U T, 0, 0, 0',
	X =  2171.990  mm,	Y =   -24.925  mm,	Z =  -336.558  mm,
	W =    -4.854 deg,	P =     4.648 deg,	R =    10.738 deg
   GP2:
	UF : 1, UT : 1,
	J1=    45.000 deg,	J2=   182.246 deg
};
P[234]{
   GP1:
	UF : 1, UT : 1,		CONFIG : 'N U T, 0, 0, 0',
	X =  2525.957  mm,	Y =  -153.860  mm,	Z =   104.179  mm,
	W =    36.503 deg,	P =    18.679 deg,	R =   -19.970 deg
   GP2:
	UF : 1, UT : 1,
	J1=    80.000 deg,	J2=    90.000 deg
};
P[235]{
   GP1:
	UF : 1, UT : 1,		CONFIG : 'N U T, 0, 0, 0',
	X =  2443.957  mm,	Y =  -153.860  mm,	Z =    41.179  mm,
	W =    36.503 deg,	P =    18.679 deg,	R =    32.647 deg
   GP2:
	UF : 1, UT : 1,
	J1=    80.000 deg,	J2=    90.000 deg
};
P[236]{
   GP1:
	UF : 1, UT : 1,		CONFIG : 'N U T, 0, 0, 0',
	X =  2224.991  mm,	Y =    21.350  mm,	Z =  -199.420  mm,
	W =   -26.754 deg,	P =    37.334 deg,	R =   139.553 deg
   GP2:
	UF : 1, UT : 1,
	J1=     0.000 deg,	J2=   180.000 deg
};
P[237]{
   GP1:
	UF : 1, UT : 1,		CONFIG : 'N U T, 0, 0, 0',
	X =  2224.989  mm,	Y =     5.850  mm,	Z =  -199.421  mm,
	W =   -26.754 deg,	P =    37.334 deg,	R =   115.158 deg
   GP2:
	UF : 1, UT : 1,
	J1=     0.000 deg,	J2=   180.000 deg
};
P[238]{
   GP1:
	UF : 1, UT : 1,		CONFIG : 'N U T, 0, 0, 0',
	X =  1476.755  mm,	Y =  -650.709  mm,	Z =     9.811  mm,
	W =    42.351 deg,	P =    16.901 deg,	R =  -100.923 deg
   GP2:
	UF : 1, UT : 1,
	J1=     0.000 deg,	J2=   180.000 deg
};
P[239]{
   GP1:
	UF : 1, UT : 1,		CONFIG : 'N U T, 0, 0, 1',
	X =  1478.206  mm,	Y =  -468.703  mm,	Z =     4.629  mm,
	W =    42.351 deg,	P =    16.901 deg,	R =  -100.923 deg
   GP2:
	UF : 1, UT : 1,
	J1=     0.000 deg,	J2=   180.000 deg
};
P[240]{
   GP1:
	UF : 1, UT : 1,		CONFIG : 'N U T, 0, 0, 0',
	X =  2443.958  mm,	Y =  -141.290  mm,	Z =    41.179  mm,
	W =    36.502 deg,	P =    18.679 deg,	R =    44.252 deg
   GP2:
	UF : 1, UT : 1,
	J1=    80.000 deg,	J2=    90.000 deg
};
P[241]{
   GP1:
	UF : 1, UT : 1,		CONFIG : 'N U T, 0, 0, 0',
	X =  2525.957  mm,	Y =  -153.860  mm,	Z =   104.179  mm,
	W =    36.503 deg,	P =    18.679 deg,	R =   -19.970 deg
   GP2:
	UF : 1, UT : 1,
	J1=    80.000 deg,	J2=    90.000 deg
};
P[242]{
   GP1:
	UF : 1, UT : 1,		CONFIG : 'N U T, 0, 0, 0',
	X =  1638.942  mm,	Y =  -220.932  mm,	Z =   176.092  mm,
	W =    39.659 deg,	P =    20.135 deg,	R =   -30.806 deg
   GP2:
	UF : 1, UT : 1,
	J1=    90.000 deg,	J2=    90.000 deg
};
P[243]{
   GP1:
	UF : 1, UT : 1,		CONFIG : 'N U T, 0, 0, 0',
	X =  1677.355  mm,	Y =  -241.647  mm,	Z =    77.021  mm,
	W =    39.659 deg,	P =    20.135 deg,	R =   -14.061 deg
   GP2:
	UF : 1, UT : 1,
	J1=    90.000 deg,	J2=    90.000 deg
};
P[244]{
   GP1:
	UF : 1, UT : 1,		CONFIG : 'N U T, 0, 0, 1',
	X =  1478.635  mm,	Y =  -447.917  mm,	Z =     4.627  mm,
	W =    42.350 deg,	P =    16.901 deg,	R =   -92.985 deg
   GP2:
	UF : 1, UT : 1,
	J1=     0.000 deg,	J2=   180.000 deg
};
P[245]{
   GP1:
	UF : 1, UT : 1,		CONFIG : 'N U T, 0, 0, 0',
	X =  1451.832  mm,	Y =     5.173  mm,	Z =     4.804  mm,
	W =     -.700 deg,	P =    41.669 deg,	R =   176.800 deg
   GP2:
	UF : 1, UT : 1,
	J1=     0.000 deg,	J2=   180.000 deg
};
P[246]{
   GP1:
	UF : 1, UT : 1,		CONFIG : 'N U T, 0, 0, 1',
	X =  1453.932  mm,	Y =  -389.816  mm,	Z =     4.113  mm,
	W =     7.653 deg,	P =    41.714 deg,	R =  -177.646 deg
   GP2:
	UF : 1, UT : 1,
	J1=     0.000 deg,	J2=   180.000 deg
};
P[247]{
   GP1:
	UF : 1, UT : 1,		CONFIG : 'N U T, 0, 0, 0',
	X =  1453.019  mm,	Y =   382.464  mm,	Z =     3.581  mm,
	W =   -18.715 deg,	P =    37.733 deg,	R =   149.445 deg
   GP2:
	UF : 1, UT : 1,
	J1=     0.000 deg,	J2=   180.000 deg
};
P[248]{
   GP1:
	UF : 1, UT : 1,		CONFIG : 'N U T, 0, 0, 0',
	X =  1961.011  mm,	Y =  -250.911  mm,	Z =    63.963  mm,
	W =    38.570 deg,	P =    15.643 deg,	R =   -37.733 deg
   GP2:
	UF : 1, UT : 1,
	J1=    90.000 deg,	J2=    90.000 deg
};
P[249]{
   GP1:
	UF : 1, UT : 1,		CONFIG : 'N U T, 0, 0, 0',
	X =  2227.011  mm,	Y =   -35.911  mm,	Z =    63.963  mm,
	W =    41.142 deg,	P =     1.290 deg,	R =    -4.650 deg
   GP2:
	UF : 1, UT : 1,
	J1=    90.000 deg,	J2=    90.000 deg
};
P[250]{
   GP1:
	UF : 1, UT : 1,		CONFIG : 'N U T, 0, 0, 0',
	X =  1451.089  mm,	Y =     4.535  mm,	Z =     3.580  mm,
	W =      .274 deg,	P =    41.491 deg,	R =   174.600 deg
   GP2:
	UF : 1, UT : 1,
	J1=     0.000 deg,	J2=   180.000 deg
};
P[251]{
   GP1:
	UF : 1, UT : 1,		CONFIG : 'N U T, 0, 0, -1',
	X =  1472.119  mm,	Y =   643.927  mm,	Z =     6.907  mm,
	W =    29.557 deg,	P =    31.284 deg,	R =  -136.748 deg
   GP2:
	UF : 1, UT : 1,
	J1=     0.000 deg,	J2=   180.000 deg
};
P[252]{
   GP1:
	UF : 1, UT : 1,		CONFIG : 'N U T, 0, 0, 0',
	X =  2193.552  mm,	Y =   -35.911  mm,	Z =    63.963  mm,
	W =    41.142 deg,	P =     1.290 deg,	R =    -4.650 deg
   GP2:
	UF : 1, UT : 1,
	J1=    90.000 deg,	J2=    90.000 deg
};
P[253]{
   GP1:
	UF : 1, UT : 1,		CONFIG : 'N U T, 0, 0, -1',
	X =  1472.491  mm,	Y =   450.907  mm,	Z =     9.385  mm,
	W =    33.887 deg,	P =    26.815 deg,	R =  -128.136 deg
   GP2:
	UF : 1, UT : 1,
	J1=     0.000 deg,	J2=   180.000 deg
};
P[254]{
   GP1:
	UF : 1, UT : 1,		CONFIG : 'N U T, 0, 0, -1',
	X =  1471.145  mm,	Y =   444.892  mm,	Z =    11.024  mm,
	W =    36.402 deg,	P =    23.004 deg,	R =  -130.111 deg
   GP2:
	UF : 1, UT : 1,
	J1=     0.000 deg,	J2=   180.000 deg
};
P[255]{
   GP1:
	UF : 1, UT : 1,		CONFIG : 'N U T, 0, 0, 0',
	X =  2180.729  mm,	Y =   -81.277  mm,	Z =  -437.708  mm,
	W =     -.956 deg,	P =    22.926 deg,	R =     1.001 deg
   GP2:
	UF : 1, UT : 1,
	J1=    45.000 deg,	J2=   180.000 deg
};
P[256]{
   GP1:
	UF : 1, UT : 1,		CONFIG : 'N U T, 0, 0, 0',
	X =  2104.646  mm,	Y =   -14.305  mm,	Z =    58.276  mm,
	W =    44.920 deg,	P =     3.025 deg,	R =    -3.029 deg
   GP2:
	UF : 1, UT : 1,
	J1=    90.000 deg,	J2=    90.000 deg
};
P[257]{
   GP1:
	UF : 1, UT : 1,		CONFIG : 'N U T, 0, 0, 0',
	X =  2176.383  mm,	Y =  -158.501  mm,	Z =  -433.497  mm,
	W =     -.953 deg,	P =    22.927 deg,	R =    22.205 deg
   GP2:
	UF : 1, UT : 1,
	J1=    45.000 deg,	J2=   180.000 deg
};
P[258]{
   GP1:
	UF : 1, UT : 1,		CONFIG : 'N U T, 0, 0, 0',
	X =  1520.748  mm,	Y =   -80.175  mm,	Z =   -54.417  mm,
	W =     5.078 deg,	P =    -9.921 deg,	R =   -27.317 deg
   GP2:
	UF : 1, UT : 1,
	J1=     0.000 deg,	J2=   180.000 deg
};
P[259]{
   GP1:
	UF : 1, UT : 1,		CONFIG : 'N U T, 0, 0, 0',
	X =  1520.919  mm,	Y =  -106.722  mm,	Z =   -58.346  mm,
	W =     5.085 deg,	P =    -9.924 deg,	R =   -27.312 deg
   GP2:
	UF : 1, UT : 1,
	J1=     0.000 deg,	J2=   180.000 deg
};
P[260]{
   GP1:
	UF : 1, UT : 1,		CONFIG : 'N U T, 0, 0, 0',
	X =  2104.646  mm,	Y =   -54.652  mm,	Z =   175.276  mm,
	W =    44.920 deg,	P =     3.025 deg,	R =    -3.029 deg
   GP2:
	UF : 1, UT : 1,
	J1=    90.000 deg,	J2=    90.000 deg
};
P[261]{
   GP1:
	UF : 1, UT : 1,		CONFIG : 'N U T, 0, 0, 0',
	X =  1705.582  mm,	Y =   -41.652  mm,	Z =   107.776  mm,
	W =    44.920 deg,	P =     3.025 deg,	R =    11.940 deg
   GP2:
	UF : 1, UT : 1,
	J1=    90.000 deg,	J2=    90.000 deg
};
P[262]{
   GP1:
	UF : 1, UT : 1,		CONFIG : 'N U T, 0, 0, 0',
	X =  1519.752  mm,	Y =  -158.457  mm,	Z =   -55.969  mm,
	W =     4.945 deg,	P =    -9.640 deg,	R =   -27.294 deg
   GP2:
	UF : 1, UT : 1,
	J1=     0.000 deg,	J2=   180.000 deg
};
P[263]{
   GP1:
	UF : 1, UT : 1,		CONFIG : 'N U T, 0, 0, 0',
	X =  1519.726  mm,	Y =  -126.578  mm,	Z =   -54.119  mm,
	W =     6.664 deg,	P =   -12.909 deg,	R =   -27.630 deg
   GP2:
	UF : 1, UT : 1,
	J1=     0.000 deg,	J2=   180.000 deg
};
P[264]{
   GP1:
	UF : 1, UT : 1,		CONFIG : 'N U T, 0, 0, 0',
	X =  2370.149  mm,	Y =   -90.588  mm,	Z =   -30.715  mm,
	W =    40.518 deg,	P =    40.131 deg,	R =    25.512 deg
   GP2:
	UF : 1, UT : 1,
	J1=    80.000 deg,	J2=    90.000 deg
};
P[265]{
   GP1:
	UF : 1, UT : 1,		CONFIG : 'N U T, 0, 0, 0',
	X =  1700.208  mm,	Y =   -40.379  mm,	Z =   119.303  mm,
	W =    53.172 deg,	P =     1.611 deg,	R =    24.177 deg
   GP2:
	UF : 1, UT : 1,
	J1=    90.000 deg,	J2=    90.000 deg
};
P[266]{
   GP1:
	UF : 1, UT : 1,		CONFIG : 'N U T, 0, 0, 0',
	X =  2369.506  mm,	Y =  -111.588  mm,	Z =   -30.715  mm,
	W =    40.518 deg,	P =    40.131 deg,	R =    53.937 deg
   GP2:
	UF : 1, UT : 1,
	J1=    80.000 deg,	J2=    90.000 deg
};
P[267]{
   GP1:
	UF : 1, UT : 1,		CONFIG : 'N U T, 0, 0, 0',
	X =  2369.507  mm,	Y =  -149.659  mm,	Z =   -30.715  mm,
	W =    40.518 deg,	P =    40.131 deg,	R =    53.937 deg
   GP2:
	UF : 1, UT : 1,
	J1=    80.000 deg,	J2=    90.000 deg
};
P[268]{
   GP1:
	UF : 1, UT : 1,		CONFIG : 'N U T, 0, 0, 0',
	X =  2368.865  mm,	Y =  -160.589  mm,	Z =   -30.715  mm,
